Universal Robots PolyScope program: mouvements camera.urp

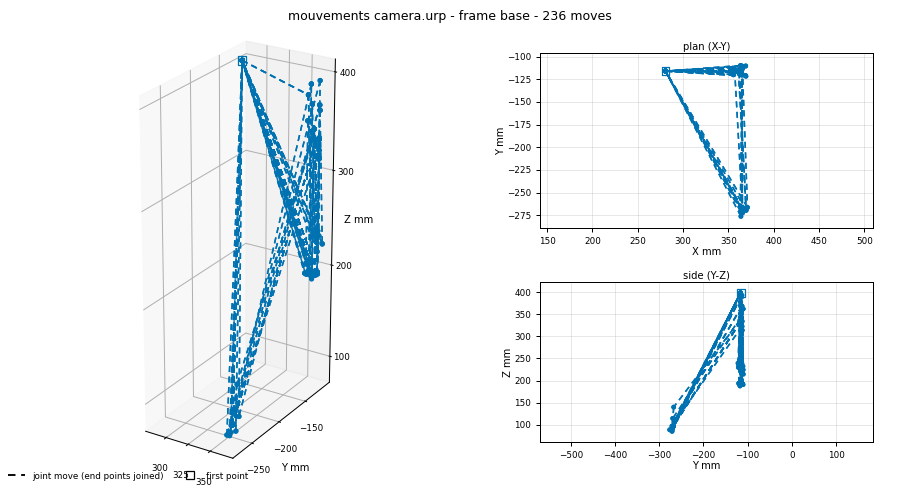
[picture p0: tool path of mouvements camera.urp in frame base, 236 of 236 moves have a stored position in this frame; points joined in program order, loops and branches not executed]
Program mouvements camera (installation=default directory=/programs/usbdisk_0 createdIn=5.21.2.0 lastSavedIn=5.12.2.1101534 robotSerialNumber=20185300595)
Calibrated DH parameters: a=[-0.000277, -0.17386, -0.213363, 0.000174, -0.000165, 0]; d=[0.151934, 52.001523, -51.96016, 0.089383, 0.08529, 0.092152]; alpha=[1.571075, 0.003287, -0.008212, 1.571169, -1.571801, 0]; deltaTheta=[0, 0.776939, 5.504669, 0.001575, 0, 0]
InitVariablesNode
Robot Program (runOnlyOnce=true)
  Folder Mouvements L'
    MoveJ speed 60 deg/s, acceleration 80 deg/s^2 (useActiveTCP=true) feature=Base
      Waypoint Waypoint_2: motionParameters(jointSpeed=1.047198 jointAcceleration=1.396263 cartesianSpeed=0.25 cartesianAcceleration=1.2); TCP in base x=280.608 y=-116.08 z=398.046 mm, rx=-2.2371 ry=2.1464 rz=-0.0359 rad; joints [2.971, -88.172, -66.4, 247.256, 90.066, 0.681] deg
      MoveJ speed 60 deg/s, acceleration 80 deg/s^2 (useActiveTCP=true) feature=Base
        Waypoint Waypoint_64: TCP in base x=354.47 y=-115.864 z=377.183 mm, rx=-3.1272 ry=-0.0242 rz=-0.0175 rad; joints [2.354, -105.869, -51.286, 247.88, 90.252, -88.495] deg
        MoveJ speed 60 deg/s, acceleration 80 deg/s^2 (useActiveTCP=true) feature=Base
          Waypoint Waypoint_65: TCP in base x=360.926 y=-115.109 z=191.362 mm, rx=-3.1273 ry=-0.0242 rz=-0.0173 rad; joints [2.478, -109.435, -98.039, 298.19, 90.28, -88.777] deg
          URCap Gripper (Robotiq_Grippers, Robotiq Inc.) dataModel(position=100.0, force=0.0, speed=0.0, positionInDouble=100.0, forceInDouble=0.0, speedInDouble=0.0, slaveIds=[2], blocking=true)
          MoveJ speed 60 deg/s, acceleration 80 deg/s^2 (useActiveTCP=true) feature=Base
            Waypoint Waypoint_66: TCP in base x=360.933 y=-115.105 z=343.669 mm, rx=-3.1273 ry=-0.0242 rz=-0.0174 rad; joints [2.446, -104.701, -62.277, 257.7, 90.221, -88.479] deg
            MoveJ speed 60 deg/s, acceleration 80 deg/s^2 (useActiveTCP=true) feature=Base
              Waypoint Waypoint_67: TCP in base x=360.932 y=-115.1 z=343.683 mm, rx=0.037 ry=-3.1303 rz=0.0223 rad; joints [2.853, -105.13, -61.17, 255.696, 88.644, 91.476] deg
              MoveJ speed 60 deg/s, acceleration 80 deg/s^2 (useActiveTCP=true) feature=Base
                Waypoint Waypoint_68: TCP in base x=369.453 y=-269.495 z=114.41 mm, rx=0.0346 ry=-2.5587 rz=-1.7903 rad; joints [-29.022, -179.68, 16.641, 199.059, 143.672, 30.692] deg
                MoveJ speed 60 deg/s, acceleration 80 deg/s^2 (useActiveTCP=true) feature=Base
                  Waypoint Waypoint_79: TCP in base x=369.462 y=-269.49 z=91.378 mm, rx=0.0347 ry=-2.5588 rz=-1.7903 rad; joints [-29.026, -184.503, 20.753, 199.764, 143.68, 30.679] deg
                URCap Gripper (Robotiq_Grippers, Robotiq Inc.) dataModel(position=0.0, force=0.0, speed=0.0, positionInDouble=0.0, forceInDouble=0.0, speedInDouble=0.0, slaveIds=[2], blocking=true)
                MoveJ speed 60 deg/s, acceleration 80 deg/s^2 (useActiveTCP=true) feature=Base
                  Waypoint Waypoint_2: motionParameters(jointSpeed=1.047198 jointAcceleration=1.396263 cartesianSpeed=0.25 cartesianAcceleration=1.2); TCP in base x=280.608 y=-116.08 z=398.046 mm, rx=-2.2371 ry=2.1464 rz=-0.0359 rad; joints [2.971, -88.172, -66.4, 247.256, 90.066, 0.681] deg
                  MoveJ speed 60 deg/s, acceleration 80 deg/s^2 (useActiveTCP=true) feature=Base
                    MoveJ speed 60 deg/s, acceleration 80 deg/s^2 (useActiveTCP=true) feature=Base
                      MoveJ speed 60 deg/s, acceleration 80 deg/s^2 (useActiveTCP=true) feature=Base
                        MoveJ speed 60 deg/s, acceleration 80 deg/s^2 (useActiveTCP=true) feature=Base
                          MoveJ speed 60 deg/s, acceleration 80 deg/s^2 (useActiveTCP=true) feature=Base
                            MoveJ speed 60 deg/s, acceleration 80 deg/s^2 (useActiveTCP=true) feature=Base
                              Waypoint Waypoint_73: TCP in base x=355.313 y=-120.114 z=193.384 mm, rx=-2.2194 ry=2.165 rz=-0.0363 rad; joints [1.736, -108.041, -100.308, 301.021, 90.164, -0.064] deg
                              URCap Gripper (Robotiq_Grippers, Robotiq Inc.) dataModel(position=100.0, force=0.0, speed=0.0, positionInDouble=100.0, forceInDouble=0.0, speedInDouble=0.0, slaveIds=[2], blocking=true)
                              MoveJ speed 60 deg/s, acceleration 80 deg/s^2 (useActiveTCP=true) feature=Base
                                Waypoint Waypoint_77: TCP in base x=355.961 y=-120.112 z=194.005 mm, rx=-3.0953 ry=0.0462 rz=0.0063 rad; joints [1.212, -108.815, -97.781, 296.498, 92.122, -87.439] deg
                                URCap Gripper (Robotiq_Grippers, Robotiq Inc.) dataModel(position=0.0, force=0.0, speed=0.0, positionInDouble=0.0, forceInDouble=0.0, speedInDouble=0.0, slaveIds=[2], blocking=true)
                                MoveJ speed 60 deg/s, acceleration 80 deg/s^2 (useActiveTCP=true) feature=Base
                                  Waypoint Waypoint_2: motionParameters(jointSpeed=1.047198 jointAcceleration=1.396263 cartesianSpeed=0.25 cartesianAcceleration=1.2); TCP in base x=280.608 y=-116.08 z=398.046 mm, rx=-2.2371 ry=2.1464 rz=-0.0359 rad; joints [2.971, -88.172, -66.4, 247.256, 90.066, 0.681] deg
                                  MoveJ speed 60 deg/s, acceleration 80 deg/s^2 (useActiveTCP=true) feature=Base
                                    Waypoint Waypoint_64: TCP in base x=354.47 y=-115.864 z=377.183 mm, rx=-3.1272 ry=-0.0242 rz=-0.0175 rad; joints [2.354, -105.869, -51.286, 247.88, 90.252, -88.495] deg
                                    MoveJ speed 60 deg/s, acceleration 80 deg/s^2 (useActiveTCP=true) feature=Base
                                      Waypoint Waypoint_65: TCP in base x=360.926 y=-115.109 z=191.362 mm, rx=-3.1273 ry=-0.0242 rz=-0.0173 rad; joints [2.478, -109.435, -98.039, 298.19, 90.28, -88.777] deg
                                      URCap Gripper (Robotiq_Grippers, Robotiq Inc.) dataModel(position=100.0, force=0.0, speed=0.0, positionInDouble=100.0, forceInDouble=0.0, speedInDouble=0.0, slaveIds=[2], blocking=true)
                                      MoveJ speed 60 deg/s, acceleration 80 deg/s^2 (useActiveTCP=true) feature=Base
                                        Waypoint Waypoint_66: TCP in base x=360.933 y=-115.105 z=343.669 mm, rx=-3.1273 ry=-0.0242 rz=-0.0174 rad; joints [2.446, -104.701, -62.277, 257.7, 90.221, -88.479] deg
                                        MoveJ speed 60 deg/s, acceleration 80 deg/s^2 (useActiveTCP=true) feature=Base
                                          Waypoint Waypoint_67: TCP in base x=360.932 y=-115.1 z=343.683 mm, rx=0.037 ry=-3.1303 rz=0.0223 rad; joints [2.853, -105.13, -61.17, 255.696, 88.644, 91.476] deg
                                          MoveJ speed 60 deg/s, acceleration 80 deg/s^2 (useActiveTCP=true) feature=Base
                                            Waypoint Waypoint_70: TCP in base x=369.313 y=-121.75 z=239.195 mm, rx=0.037 ry=-3.1302 rz=0.0223 rad; joints [1.772, -107.864, -85.879, 283.154, 88.636, 90.168] deg
                                            URCap Gripper (Robotiq_Grippers, Robotiq Inc.) dataModel(position=0.0, force=0.0, speed=0.0, positionInDouble=0.0, forceInDouble=0.0, speedInDouble=0.0, slaveIds=[2], blocking=true)
                                            MoveJ speed 60 deg/s, acceleration 80 deg/s^2 (useActiveTCP=true) feature=Base
                                              Waypoint Waypoint_2: motionParameters(jointSpeed=1.047198 jointAcceleration=1.396263 cartesianSpeed=0.25 cartesianAcceleration=1.2); TCP in base x=280.608 y=-116.08 z=398.046 mm, rx=-2.2371 ry=2.1464 rz=-0.0359 rad; joints [2.971, -88.172, -66.4, 247.256, 90.066, 0.681] deg
                                              MoveJ speed 60 deg/s, acceleration 80 deg/s^2 (useActiveTCP=true) feature=Base
                                                Waypoint Waypoint_71: TCP in base x=355.772 y=-117.714 z=191.403 mm, rx=-2.2393 ry=2.1483 rz=-0.0407 rad; joints [2.184, -108.169, -100.734, 301.575, 89.944, -0.582] deg
                                                URCap Gripper (Robotiq_Grippers, Robotiq Inc.) dataModel(position=100.0, force=0.0, speed=0.0, positionInDouble=100.0, forceInDouble=0.0, speedInDouble=0.0, slaveIds=[2], blocking=true)
                                                URCap Gripper (Robotiq_Grippers, Robotiq Inc.) dataModel(position=0.0, force=0.0, speed=0.0, positionInDouble=0.0, forceInDouble=0.0, speedInDouble=0.0, slaveIds=[2], blocking=true)
                                                MoveJ speed 60 deg/s, acceleration 80 deg/s^2 (useActiveTCP=true) feature=Base
                                                  Waypoint Waypoint_72: TCP in base x=361.681 y=-117.4 z=187.816 mm, rx=-3.1346 ry=0.019 rz=0.0078 rad; joints [2.202, -110.258, -97.51, 297.556, 89.9, -87.472] deg
                                                  URCap Gripper (Robotiq_Grippers, Robotiq Inc.) dataModel(position=100.0, force=0.0, speed=0.0, positionInDouble=100.0, forceInDouble=0.0, speedInDouble=0.0, slaveIds=[2], blocking=true)
                                                  MoveJ speed 60 deg/s, acceleration 80 deg/s^2 (useActiveTCP=true) feature=Base
                                                    Waypoint Waypoint_75: TCP in base x=361.669 y=-117.405 z=336.568 mm, rx=-3.1346 ry=0.0189 rz=0.0078 rad; joints [2.169, -105.101, -63.323, 258.214, 89.842, -87.187] deg
                                                    MoveJ speed 60 deg/s, acceleration 80 deg/s^2 (useActiveTCP=true) feature=Base
                                                      Waypoint Waypoint_76: TCP in base x=369.461 y=-267.242 z=139.99 mm, rx=-1.9057 ry=0.0195 rz=0.0548 rad; joints [-28.823, -170.798, 4.334, 201.346, 144.189, -147.418] deg
                                                      MoveJ speed 60 deg/s, acceleration 80 deg/s^2 (useActiveTCP=true) feature=Base
                                                        Waypoint Waypoint_78: TCP in base x=363.434 y=-271.007 z=85.521 mm, rx=-1.8332 ry=0.0118 rz=0.0275 rad; joints [-29.831, -179.351, 7.546, 200.182, 146.023, -154.193] deg
                                                        Waypoint Waypoint_78: TCP in base x=363.434 y=-271.007 z=85.521 mm, rx=-1.8332 ry=0.0118 rz=0.0275 rad; joints [-29.831, -179.351, 7.546, 200.182, 146.023, -154.193] deg
                                                      URCap Gripper (Robotiq_Grippers, Robotiq Inc.) dataModel(position=0.0, force=0.0, speed=0.0, positionInDouble=0.0, forceInDouble=0.0, speedInDouble=0.0, slaveIds=[2], blocking=true)
                                                      MoveJ speed 60 deg/s, acceleration 80 deg/s^2 (useActiveTCP=true) feature=Base
                                                        Waypoint Waypoint_2: motionParameters(jointSpeed=1.047198 jointAcceleration=1.396263 cartesianSpeed=0.25 cartesianAcceleration=1.2); TCP in base x=280.608 y=-116.08 z=398.046 mm, rx=-2.2371 ry=2.1464 rz=-0.0359 rad; joints [2.971, -88.172, -66.4, 247.256, 90.066, 0.681] deg
  Folder Mouvements L
    MoveJ speed 60 deg/s, acceleration 80 deg/s^2 (useActiveTCP=true) feature=Base
      Waypoint Waypoint_2: motionParameters(jointSpeed=1.047198 jointAcceleration=1.396263 cartesianSpeed=0.25 cartesianAcceleration=1.2); TCP in base x=280.608 y=-116.08 z=398.046 mm, rx=-2.2371 ry=2.1464 rz=-0.0359 rad; joints [2.971, -88.172, -66.4, 247.256, 90.066, 0.681] deg
      MoveJ speed 60 deg/s, acceleration 80 deg/s^2 (useActiveTCP=true) feature=Base
        Waypoint Waypoint_64: TCP in base x=354.47 y=-115.864 z=377.183 mm, rx=-3.1272 ry=-0.0242 rz=-0.0175 rad; joints [2.354, -105.869, -51.286, 247.88, 90.252, -88.495] deg
        MoveJ speed 60 deg/s, acceleration 80 deg/s^2 (useActiveTCP=true) feature=Base
          Waypoint Waypoint_65: TCP in base x=360.926 y=-115.109 z=191.362 mm, rx=-3.1273 ry=-0.0242 rz=-0.0173 rad; joints [2.478, -109.435, -98.039, 298.19, 90.28, -88.777] deg
          URCap Gripper (Robotiq_Grippers, Robotiq Inc.) dataModel(position=100.0, force=0.0, speed=0.0, positionInDouble=100.0, forceInDouble=0.0, speedInDouble=0.0, slaveIds=[2], blocking=true)
          MoveJ speed 60 deg/s, acceleration 80 deg/s^2 (useActiveTCP=true) feature=Base
            Waypoint Waypoint_66: TCP in base x=360.933 y=-115.105 z=343.669 mm, rx=-3.1273 ry=-0.0242 rz=-0.0174 rad; joints [2.446, -104.701, -62.277, 257.7, 90.221, -88.479] deg
            MoveJ speed 60 deg/s, acceleration 80 deg/s^2 (useActiveTCP=true) feature=Base
              Waypoint Waypoint_67: TCP in base x=360.932 y=-115.1 z=343.683 mm, rx=0.037 ry=-3.1303 rz=0.0223 rad; joints [2.853, -105.13, -61.17, 255.696, 88.644, 91.476] deg
              MoveJ speed 60 deg/s, acceleration 80 deg/s^2 (useActiveTCP=true) feature=Base
                Waypoint Waypoint_68: TCP in base x=369.453 y=-269.495 z=114.41 mm, rx=0.0346 ry=-2.5587 rz=-1.7903 rad; joints [-29.022, -179.68, 16.641, 199.059, 143.672, 30.692] deg
                MoveJ speed 60 deg/s, acceleration 80 deg/s^2 (useActiveTCP=true) feature=Base
                  Waypoint Waypoint_79: TCP in base x=369.462 y=-269.49 z=91.378 mm, rx=0.0347 ry=-2.5588 rz=-1.7903 rad; joints [-29.026, -184.503, 20.753, 199.764, 143.68, 30.679] deg
                URCap Gripper (Robotiq_Grippers, Robotiq Inc.) dataModel(position=0.0, force=0.0, speed=0.0, positionInDouble=0.0, forceInDouble=0.0, speedInDouble=0.0, slaveIds=[2], blocking=true)
                MoveJ speed 60 deg/s, acceleration 80 deg/s^2 (useActiveTCP=true) feature=Base
                  Waypoint Waypoint_2: motionParameters(jointSpeed=1.047198 jointAcceleration=1.396263 cartesianSpeed=0.25 cartesianAcceleration=1.2); TCP in base x=280.608 y=-116.08 z=398.046 mm, rx=-2.2371 ry=2.1464 rz=-0.0359 rad; joints [2.971, -88.172, -66.4, 247.256, 90.066, 0.681] deg
                  MoveJ speed 60 deg/s, acceleration 80 deg/s^2 (useActiveTCP=true) feature=Base
                    MoveJ speed 60 deg/s, acceleration 80 deg/s^2 (useActiveTCP=true) feature=Base
                      MoveJ speed 60 deg/s, acceleration 80 deg/s^2 (useActiveTCP=true) feature=Base
                        MoveJ speed 60 deg/s, acceleration 80 deg/s^2 (useActiveTCP=true) feature=Base
                          MoveJ speed 60 deg/s, acceleration 80 deg/s^2 (useActiveTCP=true) feature=Base
                            Waypoint Waypoint_2: motionParameters(jointSpeed=1.047198 jointAcceleration=1.396263 cartesianSpeed=0.25 cartesianAcceleration=1.2); TCP in base x=280.608 y=-116.08 z=398.046 mm, rx=-2.2371 ry=2.1464 rz=-0.0359 rad; joints [2.971, -88.172, -66.4, 247.256, 90.066, 0.681] deg
                            MoveJ speed 60 deg/s, acceleration 80 deg/s^2 (useActiveTCP=true) feature=Base
                              Waypoint Waypoint_73: TCP in base x=355.313 y=-120.114 z=193.384 mm, rx=-2.2194 ry=2.165 rz=-0.0363 rad; joints [1.736, -108.041, -100.308, 301.021, 90.164, -0.064] deg
                              URCap Gripper (Robotiq_Grippers, Robotiq Inc.) dataModel(position=100.0, force=0.0, speed=0.0, positionInDouble=100.0, forceInDouble=0.0, speedInDouble=0.0, slaveIds=[2], blocking=true)
                              MoveJ speed 60 deg/s, acceleration 80 deg/s^2 (useActiveTCP=true) feature=Base
                                Waypoint Waypoint_74: TCP in base x=354.955 y=-112.49 z=193.442 mm, rx=-0.1703 ry=3.1218 rz=-0.0705 rad; joints [3.842, -107.298, -100.501, 298.663, 86.895, 87.201] deg
                                URCap Gripper (Robotiq_Grippers, Robotiq Inc.) dataModel(position=0.0, force=0.0, speed=0.0, positionInDouble=0.0, forceInDouble=0.0, speedInDouble=0.0, slaveIds=[2], blocking=true)
                                MoveJ speed 60 deg/s, acceleration 80 deg/s^2 (useActiveTCP=true) feature=Base
                                  Waypoint Waypoint_2: motionParameters(jointSpeed=1.047198 jointAcceleration=1.396263 cartesianSpeed=0.25 cartesianAcceleration=1.2); TCP in base x=280.608 y=-116.08 z=398.046 mm, rx=-2.2371 ry=2.1464 rz=-0.0359 rad; joints [2.971, -88.172, -66.4, 247.256, 90.066, 0.681] deg
                                  MoveJ speed 60 deg/s, acceleration 80 deg/s^2 (useActiveTCP=true) feature=Base
                                    Waypoint Waypoint_64: TCP in base x=354.47 y=-115.864 z=377.183 mm, rx=-3.1272 ry=-0.0242 rz=-0.0175 rad; joints [2.354, -105.869, -51.286, 247.88, 90.252, -88.495] deg
                                    MoveJ speed 60 deg/s, acceleration 80 deg/s^2 (useActiveTCP=true) feature=Base
                                      Waypoint Waypoint_65: TCP in base x=360.926 y=-115.109 z=191.362 mm, rx=-3.1273 ry=-0.0242 rz=-0.0173 rad; joints [2.478, -109.435, -98.039, 298.19, 90.28, -88.777] deg
                                      URCap Gripper (Robotiq_Grippers, Robotiq Inc.) dataModel(position=100.0, force=0.0, speed=0.0, positionInDouble=100.0, forceInDouble=0.0, speedInDouble=0.0, slaveIds=[2], blocking=true)
                                      MoveJ speed 60 deg/s, acceleration 80 deg/s^2 (useActiveTCP=true) feature=Base
                                        Waypoint Waypoint_66: TCP in base x=360.933 y=-115.105 z=343.669 mm, rx=-3.1273 ry=-0.0242 rz=-0.0174 rad; joints [2.446, -104.701, -62.277, 257.7, 90.221, -88.479] deg
                                        MoveJ speed 60 deg/s, acceleration 80 deg/s^2 (useActiveTCP=true) feature=Base
                                          Waypoint Waypoint_67: TCP in base x=360.932 y=-115.1 z=343.683 mm, rx=0.037 ry=-3.1303 rz=0.0223 rad; joints [2.853, -105.13, -61.17, 255.696, 88.644, 91.476] deg
                                          MoveJ speed 60 deg/s, acceleration 80 deg/s^2 (useActiveTCP=true) feature=Base
                                            Waypoint Waypoint_70: TCP in base x=369.313 y=-121.75 z=239.195 mm, rx=0.037 ry=-3.1302 rz=0.0223 rad; joints [1.772, -107.864, -85.879, 283.154, 88.636, 90.168] deg
                                            URCap Gripper (Robotiq_Grippers, Robotiq Inc.) dataModel(position=0.0, force=0.0, speed=0.0, positionInDouble=0.0, forceInDouble=0.0, speedInDouble=0.0, slaveIds=[2], blocking=true)
                                            MoveJ speed 60 deg/s, acceleration 80 deg/s^2 (useActiveTCP=true) feature=Base
                                              Waypoint Waypoint_2: motionParameters(jointSpeed=1.047198 jointAcceleration=1.396263 cartesianSpeed=0.25 cartesianAcceleration=1.2); TCP in base x=280.608 y=-116.08 z=398.046 mm, rx=-2.2371 ry=2.1464 rz=-0.0359 rad; joints [2.971, -88.172, -66.4, 247.256, 90.066, 0.681] deg
                                              MoveJ speed 60 deg/s, acceleration 80 deg/s^2 (useActiveTCP=true) feature=Base
                                                Waypoint Waypoint_71: TCP in base x=355.772 y=-117.714 z=191.403 mm, rx=-2.2393 ry=2.1483 rz=-0.0407 rad; joints [2.184, -108.169, -100.734, 301.575, 89.944, -0.582] deg
                                                URCap Gripper (Robotiq_Grippers, Robotiq Inc.) dataModel(position=100.0, force=0.0, speed=0.0, positionInDouble=100.0, forceInDouble=0.0, speedInDouble=0.0, slaveIds=[2], blocking=true)
                                                URCap Gripper (Robotiq_Grippers, Robotiq Inc.) dataModel(position=0.0, force=0.0, speed=0.0, positionInDouble=0.0, forceInDouble=0.0, speedInDouble=0.0, slaveIds=[2], blocking=true)
                                                MoveJ speed 60 deg/s, acceleration 80 deg/s^2 (useActiveTCP=true) feature=Base
                                                  Waypoint Waypoint_72: TCP in base x=361.681 y=-117.4 z=187.816 mm, rx=-3.1346 ry=0.019 rz=0.0078 rad; joints [2.202, -110.258, -97.51, 297.556, 89.9, -87.472] deg
                                                  URCap Gripper (Robotiq_Grippers, Robotiq Inc.) dataModel(position=100.0, force=0.0, speed=0.0, positionInDouble=100.0, forceInDouble=0.0, speedInDouble=0.0, slaveIds=[2], blocking=true)
                                                  MoveJ speed 60 deg/s, acceleration 80 deg/s^2 (useActiveTCP=true) feature=Base
                                                    Waypoint Waypoint_75: TCP in base x=361.669 y=-117.405 z=336.568 mm, rx=-3.1346 ry=0.0189 rz=0.0078 rad; joints [2.169, -105.101, -63.323, 258.214, 89.842, -87.187] deg
                                                    MoveJ speed 60 deg/s, acceleration 80 deg/s^2 (useActiveTCP=true) feature=Base
                                                      Waypoint Waypoint_76: TCP in base x=369.461 y=-267.242 z=139.99 mm, rx=-1.9057 ry=0.0195 rz=0.0548 rad; joints [-28.823, -170.798, 4.334, 201.346, 144.189, -147.418] deg
                                                      MoveJ speed 60 deg/s, acceleration 80 deg/s^2 (useActiveTCP=true) feature=Base
                                                        Waypoint Waypoint_78: TCP in base x=363.434 y=-271.007 z=85.521 mm, rx=-1.8332 ry=0.0118 rz=0.0275 rad; joints [-29.831, -179.351, 7.546, 200.182, 146.023, -154.193] deg
                                                      URCap Gripper (Robotiq_Grippers, Robotiq Inc.) dataModel(position=0.0, force=0.0, speed=0.0, positionInDouble=0.0, forceInDouble=0.0, speedInDouble=0.0, slaveIds=[2], blocking=true)
                                                      MoveJ speed 60 deg/s, acceleration 80 deg/s^2 (useActiveTCP=true) feature=Base
                                                        Waypoint Waypoint_2: motionParameters(jointSpeed=1.047198 jointAcceleration=1.396263 cartesianSpeed=0.25 cartesianAcceleration=1.2); TCP in base x=280.608 y=-116.08 z=398.046 mm, rx=-2.2371 ry=2.1464 rz=-0.0359 rad; joints [2.971, -88.172, -66.4, 247.256, 90.066, 0.681] deg
  Folder Mouvement U
    MoveJ speed 60 deg/s, acceleration 80 deg/s^2 (useActiveTCP=true) feature=Base
      Waypoint Waypoint_2: motionParameters(jointSpeed=1.047198 jointAcceleration=1.396263 cartesianSpeed=0.25 cartesianAcceleration=1.2); TCP in base x=280.608 y=-116.08 z=398.046 mm, rx=-2.2371 ry=2.1464 rz=-0.0359 rad; joints [2.971, -88.172, -66.4, 247.256, 90.066, 0.681] deg
      MoveJ speed 60 deg/s, acceleration 80 deg/s^2 (useActiveTCP=true) feature=Base
        Waypoint Waypoint_8: TCP in base x=360.359 y=-116.083 z=194.377 mm, rx=-2.248 ry=2.1578 rz=0.0022 rad; joints [2.251, -109.03, -97.858, 297.936, 90.564, -0.456] deg
        URCap Gripper (Robotiq_Grippers, Robotiq Inc.) dataModel(position=100.0, force=0.0, speed=0.0, positionInDouble=100.0, forceInDouble=0.0, speedInDouble=0.0, slaveIds=[2], blocking=true)
        MoveJ speed 60 deg/s, acceleration 80 deg/s^2 (useActiveTCP=true) feature=Base
          Waypoint Waypoint_11: TCP in base x=360.347 y=-116.075 z=194.373 mm, rx=-0.1344 ry=3.1191 rz=-0.0257 rad; joints [2.778, -108.754, -98.304, 298.232, 88.541, 87.461] deg
          URCap Gripper (Robotiq_Grippers, Robotiq Inc.) dataModel(position=0.0, force=0.0, speed=0.0, positionInDouble=0.0, forceInDouble=0.0, speedInDouble=0.0, slaveIds=[2], blocking=true)
          MoveJ speed 60 deg/s, acceleration 80 deg/s^2 (useActiveTCP=true) feature=Base
            Waypoint Waypoint_2: motionParameters(jointSpeed=1.047198 jointAcceleration=1.396263 cartesianSpeed=0.25 cartesianAcceleration=1.2); TCP in base x=280.608 y=-116.08 z=398.046 mm, rx=-2.2371 ry=2.1464 rz=-0.0359 rad; joints [2.971, -88.172, -66.4, 247.256, 90.066, 0.681] deg
          Folder Mouvement U'
            MoveJ speed 60 deg/s, acceleration 80 deg/s^2 (useActiveTCP=true) feature=Base
              Waypoint Waypoint_2: motionParameters(jointSpeed=1.047198 jointAcceleration=1.396263 cartesianSpeed=0.25 cartesianAcceleration=1.2); TCP in base x=280.608 y=-116.08 z=398.046 mm, rx=-2.2371 ry=2.1464 rz=-0.0359 rad; joints [2.971, -88.172, -66.4, 247.256, 90.066, 0.681] deg
              MoveJ speed 60 deg/s, acceleration 80 deg/s^2 (useActiveTCP=true) feature=Base
                Waypoint Waypoint_13: TCP in base x=360.129 y=-115.918 z=194.945 mm, rx=-2.246 ry=2.1551 rz=-0.0175 rad; joints [2.383, -108.75, -98.377, 298.822, 90.174, -0.353] deg
                URCap Gripper (Robotiq_Grippers, Robotiq Inc.) dataModel(position=100.0, force=0.0, speed=0.0, positionInDouble=100.0, forceInDouble=0.0, speedInDouble=0.0, slaveIds=[2], blocking=true)
                MoveJ speed 60 deg/s, acceleration 80 deg/s^2 (useActiveTCP=true) feature=Base
                  Waypoint Waypoint_12: TCP in base x=360.146 y=-115.908 z=194.96 mm, rx=-3.1124 ry=-0.0686 rz=0.0193 rad; joints [2.131, -109.287, -96.569, 295.219, 91.114, -90.75] deg
                  URCap Gripper (Robotiq_Grippers, Robotiq Inc.) dataModel(position=0.0, force=0.0, speed=0.0, positionInDouble=0.0, forceInDouble=0.0, speedInDouble=0.0, slaveIds=[2], blocking=true)
                  Folder Mouvement F
                    MoveJ speed 60 deg/s, acceleration 80 deg/s^2 (useActiveTCP=true) feature=Base
                      Waypoint Waypoint_2: motionParameters(jointSpeed=1.047198 jointAcceleration=1.396263 cartesianSpeed=0.25 cartesianAcceleration=1.2); TCP in base x=280.608 y=-116.08 z=398.046 mm, rx=-2.2371 ry=2.1464 rz=-0.0359 rad; joints [2.971, -88.172, -66.4, 247.256, 90.066, 0.681] deg
                      MoveJ speed 60 deg/s, acceleration 80 deg/s^2 (useActiveTCP=true) feature=Base
                        Waypoint Waypoint_14: TCP in base x=365.369 y=-113.056 z=194.065 mm, rx=-2.2548 ry=2.1638 rz=0.001 rad; joints [2.803, -109.941, -96.5, 297.16, 90.168, 0.082] deg
                        URCap Gripper (Robotiq_Grippers, Robotiq Inc.) dataModel(position=100.0, force=0.0, speed=0.0, positionInDouble=100.0, forceInDouble=0.0, speedInDouble=0.0, slaveIds=[2], blocking=true)
                        MoveJ speed 60 deg/s, acceleration 80 deg/s^2 (useActiveTCP=true) feature=Base
                          Waypoint Waypoint_15: TCP in base x=365.367 y=-113.056 z=313.339 mm, rx=-2.2546 ry=2.1637 rz=0.001 rad; joints [2.778, -104.495, -70.787, 266.006, 90.105, 0.314] deg
                          MoveJ speed 60 deg/s, acceleration 80 deg/s^2 (useActiveTCP=true) feature=Base
                            Waypoint Waypoint_23: TCP in base x=365.372 y=-113.061 z=392.746 mm, rx=-3.1299 ry=0.0024 rz=0.0189 rad; joints [2.738, -112.179, -37.095, 238.673, 90.207, -87.085] deg
                          MoveJ speed 60 deg/s, acceleration 80 deg/s^2 (useActiveTCP=true) feature=Base
                            Waypoint Waypoint_16: TCP in base x=363.126 y=-264.93 z=106.645 mm, rx=-1.9305 ry=-0.0066 rz=-0.0141 rad; joints [-29.004, -157.4, -33.157, 229.064, 144.815, -147.561] deg
                            URCap Gripper (Robotiq_Grippers, Robotiq Inc.) dataModel(position=0.0, force=0.0, speed=0.0, positionInDouble=0.0, forceInDouble=0.0, speedInDouble=0.0, slaveIds=[2], blocking=true)
                            MoveJ speed 60 deg/s, acceleration 80 deg/s^2 (useActiveTCP=true) feature=Base
                              Waypoint Waypoint_2: motionParameters(jointSpeed=1.047198 jointAcceleration=1.396263 cartesianSpeed=0.25 cartesianAcceleration=1.2); TCP in base x=280.608 y=-116.08 z=398.046 mm, rx=-2.2371 ry=2.1464 rz=-0.0359 rad; joints [2.971, -88.172, -66.4, 247.256, 90.066, 0.681] deg
                              MoveJ speed 60 deg/s, acceleration 80 deg/s^2 (useActiveTCP=true) feature=Base
                                Waypoint Waypoint_17: TCP in base x=359.006 y=-116.088 z=193.011 mm, rx=-2.2371 ry=2.1464 rz=-0.0359 rad; joints [2.365, -108.587, -99.655, 300.918, 90.181, -0.384] deg
                                URCap Gripper (Robotiq_Grippers, Robotiq Inc.) dataModel(position=100.0, force=0.0, speed=0.0, positionInDouble=100.0, forceInDouble=0.0, speedInDouble=0.0, slaveIds=[2], blocking=true)
                                MoveJ speed 60 deg/s, acceleration 80 deg/s^2 (useActiveTCP=true) feature=Base
                                  Waypoint Waypoint_18: TCP in base x=359.004 y=-116.091 z=368.94 mm, rx=-2.2371 ry=2.1464 rz=-0.0359 rad; joints [2.326, -105.125, -55.5, 253.299, 90.124, -0.043] deg
                                  MoveJ speed 60 deg/s, acceleration 80 deg/s^2 (useActiveTCP=true) feature=Base
                                    Waypoint Waypoint_19: TCP in base x=359.011 y=-116.091 z=368.946 mm, rx=-3.0949 ry=-0.0873 rz=0.0203 rad; joints [1.817, -107.4, -51.023, 247.739, 92.062, -91.397] deg
                                    MoveJ speed 60 deg/s, acceleration 80 deg/s^2 (useActiveTCP=true) feature=Base
                                      Waypoint Waypoint_20: TCP in base x=366.237 y=-120.423 z=235.896 mm, rx=-3.0949 ry=-0.0874 rz=0.0204 rad; joints [1.134, -107.736, -86.938, 283.944, 92.035, -92.376] deg
                                      URCap Gripper (Robotiq_Grippers, Robotiq Inc.) dataModel(position=0.0, force=0.0, speed=0.0, positionInDouble=0.0, forceInDouble=0.0, speedInDouble=0.0, slaveIds=[2], blocking=true)
                                      MoveJ speed 60 deg/s, acceleration 80 deg/s^2 (useActiveTCP=true) feature=Base
                                        Waypoint Waypoint_2: motionParameters(jointSpeed=1.047198 jointAcceleration=1.396263 cartesianSpeed=0.25 cartesianAcceleration=1.2); TCP in base x=280.608 y=-116.08 z=398.046 mm, rx=-2.2371 ry=2.1464 rz=-0.0359 rad; joints [2.971, -88.172, -66.4, 247.256, 90.066, 0.681] deg
                                        MoveJ speed 60 deg/s, acceleration 80 deg/s^2 (useActiveTCP=true) feature=Base
                                          Waypoint Waypoint_21: TCP in base x=364.127 y=-117.777 z=193.293 mm, rx=-2.2569 ry=2.1661 rz=0.0165 rad; joints [1.986, -110.209, -96.105, 296.494, 90.452, -0.727] deg
                                          URCap Gripper (Robotiq_Grippers, Robotiq Inc.) dataModel(position=100.0, force=0.0, speed=0.0, positionInDouble=100.0, forceInDouble=0.0, speedInDouble=0.0, slaveIds=[2], blocking=true)
                                          MoveJ speed 60 deg/s, acceleration 80 deg/s^2 (useActiveTCP=true) feature=Base
                                            Waypoint Waypoint_32: TCP in base x=364.117 y=-117.792 z=193.289 mm, rx=-0.0015 ry=3.1247 rz=-0.0036 rad; joints [2.276, -109.92, -96.897, 297.836, 89.322, 91.847] deg
                                          MoveJ speed 60 deg/s, acceleration 80 deg/s^2 (useActiveTCP=true) feature=Base
                                            MoveJ speed 60 deg/s, acceleration 80 deg/s^2 (useActiveTCP=true) feature=Base
                                              Waypoint Waypoint_2: motionParameters(jointSpeed=1.047198 jointAcceleration=1.396263 cartesianSpeed=0.25 cartesianAcceleration=1.2); TCP in base x=280.608 y=-116.08 z=398.046 mm, rx=-2.2371 ry=2.1464 rz=-0.0359 rad; joints [2.971, -88.172, -66.4, 247.256, 90.066, 0.681] deg
                                              MoveJ speed 60 deg/s, acceleration 80 deg/s^2 (useActiveTCP=true) feature=Base
                                                Waypoint Waypoint_24: TCP in base x=356.858 y=-114.748 z=193.459 mm, rx=-2.237 ry=2.1464 rz=-0.0359 rad; joints [2.599, -107.985, -100.366, 301.027, 90.17, -0.146] deg
                                                URCap Gripper (Robotiq_Grippers, Robotiq Inc.) dataModel(position=100.0, force=0.0, speed=0.0, positionInDouble=100.0, forceInDouble=0.0, speedInDouble=0.0, slaveIds=[2], blocking=true)
                                                MoveJ speed 60 deg/s, acceleration 80 deg/s^2 (useActiveTCP=true) feature=Base
                                                  Waypoint Waypoint_25: TCP in base x=356.855 y=-114.738 z=388.235 mm, rx=-2.2372 ry=2.1464 rz=-0.0359 rad; joints [2.556, -106.57, -47.975, 247.22, 90.134, 0.231] deg
                                                  MoveJ speed 60 deg/s, acceleration 80 deg/s^2 (useActiveTCP=true) feature=Base
                                                    Waypoint Waypoint_27: TCP in base x=356.863 y=-114.749 z=388.208 mm, rx=-3.1012 ry=-0.0612 rz=0.0211 rad; joints [2.118, -109.149, -42.896, 241.364, 91.775, -90.078] deg
                                                  MoveJ speed 60 deg/s, acceleration 80 deg/s^2 (useActiveTCP=true) feature=Base
                                                    Waypoint Waypoint_26: TCP in base x=365.655 y=-272.422 z=90.213 mm, rx=-1.8494 ry=-0.0463 rz=-0.0141 rad; joints [-29.785, -175.347, 0.325, 204.9, 145.531, -156.47] deg
                                                    URCap Gripper (Robotiq_Grippers, Robotiq Inc.) dataModel(position=0.0, force=0.0, speed=0.0, positionInDouble=0.0, forceInDouble=0.0, speedInDouble=0.0, slaveIds=[2], blocking=true)
                                                    MoveJ speed 60 deg/s, acceleration 80 deg/s^2 (useActiveTCP=true) feature=Base
                                                      Waypoint Waypoint_2: motionParameters(jointSpeed=1.047198 jointAcceleration=1.396263 cartesianSpeed=0.25 cartesianAcceleration=1.2); TCP in base x=280.608 y=-116.08 z=398.046 mm, rx=-2.2371 ry=2.1464 rz=-0.0359 rad; joints [2.971, -88.172, -66.4, 247.256, 90.066, 0.681] deg
                                                      MoveJ speed 60 deg/s, acceleration 80 deg/s^2 (useActiveTCP=true) feature=Base
                                                        Waypoint Waypoint_28: TCP in base x=354.352 y=-116.082 z=201.505 mm, rx=-2.237 ry=2.1464 rz=-0.0359 rad; joints [2.395, -106.647, -99.774, 299.096, 90.165, -0.336] deg
                                                        URCap Gripper (Robotiq_Grippers, Robotiq Inc.) dataModel(position=100.0, force=0.0, speed=0.0, positionInDouble=100.0, forceInDouble=0.0, speedInDouble=0.0, slaveIds=[2], blocking=true)
                                                        MoveJ speed 60 deg/s, acceleration 80 deg/s^2 (useActiveTCP=true) feature=Base
                                                          Waypoint Waypoint_29: TCP in base x=354.342 y=-116.082 z=351.047 mm, rx=-2.2371 ry=2.1464 rz=-0.0359 rad; joints [2.364, -102.529, -63.836, 259.041, 90.104, -0.046] deg
                                                          MoveJ speed 60 deg/s, acceleration 80 deg/s^2 (useActiveTCP=true) feature=Base
                                                            Waypoint Waypoint_30: TCP in base x=354.353 y=-116.08 z=351.019 mm, rx=-3.0948 ry=-0.093 rz=0.0205 rad; joints [1.85, -104.53, -59.905, 253.739, 92.034, -91.617] deg
                                                            MoveJ speed 60 deg/s, acceleration 80 deg/s^2 (useActiveTCP=true) feature=Base
                                                              Waypoint Waypoint_31: TCP in base x=368.984 y=-120.916 z=229.682 mm, rx=-3.0957 ry=0.0142 rz=0.018 rad; joints [1.041, -108.753, -87.348, 285.539, 92.083, -88.72] deg
                                                              URCap Gripper (Robotiq_Grippers, Robotiq Inc.) dataModel(position=0.0, force=0.0, speed=0.0, positionInDouble=0.0, forceInDouble=0.0, speedInDouble=0.0, slaveIds=[2], blocking=true)
                                                              MoveJ speed 60 deg/s, acceleration 80 deg/s^2 (useActiveTCP=true) feature=Base
                                                                Waypoint Waypoint_2: motionParameters(jointSpeed=1.047198 jointAcceleration=1.396263 cartesianSpeed=0.25 cartesianAcceleration=1.2); TCP in base x=280.608 y=-116.08 z=398.046 mm, rx=-2.2371 ry=2.1464 rz=-0.0359 rad; joints [2.971, -88.172, -66.4, 247.256, 90.066, 0.681] deg
                  Folder Mouvement F'
                    MoveJ speed 60 deg/s, acceleration 80 deg/s^2 (useActiveTCP=true) feature=Base
                      Waypoint Waypoint_2: motionParameters(jointSpeed=1.047198 jointAcceleration=1.396263 cartesianSpeed=0.25 cartesianAcceleration=1.2); TCP in base x=280.608 y=-116.08 z=398.046 mm, rx=-2.2371 ry=2.1464 rz=-0.0359 rad; joints [2.971, -88.172, -66.4, 247.256, 90.066, 0.681] deg
                      MoveJ speed 60 deg/s, acceleration 80 deg/s^2 (useActiveTCP=true) feature=Base
                        Waypoint Waypoint_14: TCP in base x=365.369 y=-113.056 z=194.065 mm, rx=-2.2548 ry=2.1638 rz=0.001 rad; joints [2.803, -109.941, -96.5, 297.16, 90.168, 0.082] deg
                        URCap Gripper (Robotiq_Grippers, Robotiq Inc.) dataModel(position=100.0, force=0.0, speed=0.0, positionInDouble=100.0, forceInDouble=0.0, speedInDouble=0.0, slaveIds=[2], blocking=true)
                        MoveJ speed 60 deg/s, acceleration 80 deg/s^2 (useActiveTCP=true) feature=Base
                          Waypoint Waypoint_15: TCP in base x=365.367 y=-113.056 z=313.339 mm, rx=-2.2546 ry=2.1637 rz=0.001 rad; joints [2.778, -104.495, -70.787, 266.006, 90.105, 0.314] deg
                          MoveJ speed 60 deg/s, acceleration 80 deg/s^2 (useActiveTCP=true) feature=Base
                            Waypoint Waypoint_23: TCP in base x=365.372 y=-113.061 z=392.746 mm, rx=-3.1299 ry=0.0024 rz=0.0189 rad; joints [2.738, -112.179, -37.095, 238.673, 90.207, -87.085] deg
                          MoveJ speed 60 deg/s, acceleration 80 deg/s^2 (useActiveTCP=true) feature=Base
                            Waypoint Waypoint_16: TCP in base x=363.126 y=-264.93 z=106.645 mm, rx=-1.9305 ry=-0.0066 rz=-0.0141 rad; joints [-29.004, -157.4, -33.157, 229.064, 144.815, -147.561] deg
                            URCap Gripper (Robotiq_Grippers, Robotiq Inc.) dataModel(position=0.0, force=0.0, speed=0.0, positionInDouble=0.0, forceInDouble=0.0, speedInDouble=0.0, slaveIds=[2], blocking=true)
                            MoveJ speed 60 deg/s, acceleration 80 deg/s^2 (useActiveTCP=true) feature=Base
                              Waypoint Waypoint_2: motionParameters(jointSpeed=1.047198 jointAcceleration=1.396263 cartesianSpeed=0.25 cartesianAcceleration=1.2); TCP in base x=280.608 y=-116.08 z=398.046 mm, rx=-2.2371 ry=2.1464 rz=-0.0359 rad; joints [2.971, -88.172, -66.4, 247.256, 90.066, 0.681] deg
                              MoveJ speed 60 deg/s, acceleration 80 deg/s^2 (useActiveTCP=true) feature=Base
                                Waypoint Waypoint_17: TCP in base x=359.006 y=-116.088 z=193.011 mm, rx=-2.2371 ry=2.1464 rz=-0.0359 rad; joints [2.365, -108.587, -99.655, 300.918, 90.181, -0.384] deg
                                URCap Gripper (Robotiq_Grippers, Robotiq Inc.) dataModel(position=100.0, force=0.0, speed=0.0, positionInDouble=100.0, forceInDouble=0.0, speedInDouble=0.0, slaveIds=[2], blocking=true)
                                MoveJ speed 60 deg/s, acceleration 80 deg/s^2 (useActiveTCP=true) feature=Base
                                  Waypoint Waypoint_18: TCP in base x=359.004 y=-116.091 z=368.94 mm, rx=-2.2371 ry=2.1464 rz=-0.0359 rad; joints [2.326, -105.125, -55.5, 253.299, 90.124, -0.043] deg
                                  MoveJ speed 60 deg/s, acceleration 80 deg/s^2 (useActiveTCP=true) feature=Base
                                    Waypoint Waypoint_19: TCP in base x=359.011 y=-116.091 z=368.946 mm, rx=-3.0949 ry=-0.0873 rz=0.0203 rad; joints [1.817, -107.4, -51.023, 247.739, 92.062, -91.397] deg
                                    MoveJ speed 60 deg/s, acceleration 80 deg/s^2 (useActiveTCP=true) feature=Base
                                      Waypoint Waypoint_20: TCP in base x=366.237 y=-120.423 z=235.896 mm, rx=-3.0949 ry=-0.0874 rz=0.0204 rad; joints [1.134, -107.736, -86.938, 283.944, 92.035, -92.376] deg
                                      URCap Gripper (Robotiq_Grippers, Robotiq Inc.) dataModel(position=0.0, force=0.0, speed=0.0, positionInDouble=0.0, forceInDouble=0.0, speedInDouble=0.0, slaveIds=[2], blocking=true)
                                      MoveJ speed 60 deg/s, acceleration 80 deg/s^2 (useActiveTCP=true) feature=Base
                                        Waypoint Waypoint_2: motionParameters(jointSpeed=1.047198 jointAcceleration=1.396263 cartesianSpeed=0.25 cartesianAcceleration=1.2); TCP in base x=280.608 y=-116.08 z=398.046 mm, rx=-2.2371 ry=2.1464 rz=-0.0359 rad; joints [2.971, -88.172, -66.4, 247.256, 90.066, 0.681] deg
                                        MoveJ speed 60 deg/s, acceleration 80 deg/s^2 (useActiveTCP=true) feature=Base
                                          Waypoint Waypoint_21: TCP in base x=364.127 y=-117.777 z=193.293 mm, rx=-2.2569 ry=2.1661 rz=0.0165 rad; joints [1.986, -110.209, -96.105, 296.494, 90.452, -0.727] deg
                                          URCap Gripper (Robotiq_Grippers, Robotiq Inc.) dataModel(position=100.0, force=0.0, speed=0.0, positionInDouble=100.0, forceInDouble=0.0, speedInDouble=0.0, slaveIds=[2], blocking=true)
                                          MoveJ speed 60 deg/s, acceleration 80 deg/s^2 (useActiveTCP=true) feature=Base
                                            Waypoint Waypoint_22: TCP in base x=364.117 y=-117.783 z=193.288 mm, rx=-3.1392 ry=-0.0124 rz=0.0265 rad; joints [2.189, -110.312, -95.473, 294.88, 89.639, -88.615] deg
                                            URCap Gripper (Robotiq_Grippers, Robotiq Inc.) dataModel(position=0.0, force=0.0, speed=0.0, positionInDouble=0.0, forceInDouble=0.0, speedInDouble=0.0, slaveIds=[2], blocking=true)
                                          MoveJ speed 60 deg/s, acceleration 80 deg/s^2 (useActiveTCP=true) feature=Base
                                            MoveJ speed 60 deg/s, acceleration 80 deg/s^2 (useActiveTCP=true) feature=Base
                                              Waypoint Waypoint_2: motionParameters(jointSpeed=1.047198 jointAcceleration=1.396263 cartesianSpeed=0.25 cartesianAcceleration=1.2); TCP in base x=280.608 y=-116.08 z=398.046 mm, rx=-2.2371 ry=2.1464 rz=-0.0359 rad; joints [2.971, -88.172, -66.4, 247.256, 90.066, 0.681] deg
                                              MoveJ speed 60 deg/s, acceleration 80 deg/s^2 (useActiveTCP=true) feature=Base
                                                Waypoint Waypoint_24: TCP in base x=356.858 y=-114.748 z=193.459 mm, rx=-2.237 ry=2.1464 rz=-0.0359 rad; joints [2.599, -107.985, -100.366, 301.027, 90.17, -0.146] deg
                                                URCap Gripper (Robotiq_Grippers, Robotiq Inc.) dataModel(position=100.0, force=0.0, speed=0.0, positionInDouble=100.0, forceInDouble=0.0, speedInDouble=0.0, slaveIds=[2], blocking=true)
                                                MoveJ speed 60 deg/s, acceleration 80 deg/s^2 (useActiveTCP=true) feature=Base
                                                  Waypoint Waypoint_25: TCP in base x=356.855 y=-114.738 z=388.235 mm, rx=-2.2372 ry=2.1464 rz=-0.0359 rad; joints [2.556, -106.57, -47.975, 247.22, 90.134, 0.231] deg
                                                  MoveJ speed 60 deg/s, acceleration 80 deg/s^2 (useActiveTCP=true) feature=Base
                                                    Waypoint Waypoint_27: TCP in base x=356.863 y=-114.749 z=388.208 mm, rx=-3.1012 ry=-0.0612 rz=0.0211 rad; joints [2.118, -109.149, -42.896, 241.364, 91.775, -90.078] deg
                                                  MoveJ speed 60 deg/s, acceleration 80 deg/s^2 (useActiveTCP=true) feature=Base
                                                    Waypoint Waypoint_26: TCP in base x=365.655 y=-272.422 z=90.213 mm, rx=-1.8494 ry=-0.0463 rz=-0.0141 rad; joints [-29.785, -175.347, 0.325, 204.9, 145.531, -156.47] deg
                                                    URCap Gripper (Robotiq_Grippers, Robotiq Inc.) dataModel(position=0.0, force=0.0, speed=0.0, positionInDouble=0.0, forceInDouble=0.0, speedInDouble=0.0, slaveIds=[2], blocking=true)
                                                    MoveJ speed 60 deg/s, acceleration 80 deg/s^2 (useActiveTCP=true) feature=Base
                                                      Waypoint Waypoint_2: motionParameters(jointSpeed=1.047198 jointAcceleration=1.396263 cartesianSpeed=0.25 cartesianAcceleration=1.2); TCP in base x=280.608 y=-116.08 z=398.046 mm, rx=-2.2371 ry=2.1464 rz=-0.0359 rad; joints [2.971, -88.172, -66.4, 247.256, 90.066, 0.681] deg
                                                      MoveJ speed 60 deg/s, acceleration 80 deg/s^2 (useActiveTCP=true) feature=Base
                                                        Waypoint Waypoint_28: TCP in base x=354.352 y=-116.082 z=201.505 mm, rx=-2.237 ry=2.1464 rz=-0.0359 rad; joints [2.395, -106.647, -99.774, 299.096, 90.165, -0.336] deg
                                                        URCap Gripper (Robotiq_Grippers, Robotiq Inc.) dataModel(position=100.0, force=0.0, speed=0.0, positionInDouble=100.0, forceInDouble=0.0, speedInDouble=0.0, slaveIds=[2], blocking=true)
                                                        MoveJ speed 60 deg/s, acceleration 80 deg/s^2 (useActiveTCP=true) feature=Base
                                                          Waypoint Waypoint_29: TCP in base x=354.342 y=-116.082 z=351.047 mm, rx=-2.2371 ry=2.1464 rz=-0.0359 rad; joints [2.364, -102.529, -63.836, 259.041, 90.104, -0.046] deg
                                                          MoveJ speed 60 deg/s, acceleration 80 deg/s^2 (useActiveTCP=true) feature=Base
                                                            Waypoint Waypoint_30: TCP in base x=354.353 y=-116.08 z=351.019 mm, rx=-3.0948 ry=-0.093 rz=0.0205 rad; joints [1.85, -104.53, -59.905, 253.739, 92.034, -91.617] deg
                                                            MoveJ speed 60 deg/s, acceleration 80 deg/s^2 (useActiveTCP=true) feature=Base
                                                              Waypoint Waypoint_31: TCP in base x=368.984 y=-120.916 z=229.682 mm, rx=-3.0957 ry=0.0142 rz=0.018 rad; joints [1.041, -108.753, -87.348, 285.539, 92.083, -88.72] deg
                                                              URCap Gripper (Robotiq_Grippers, Robotiq Inc.) dataModel(position=0.0, force=0.0, speed=0.0, positionInDouble=0.0, forceInDouble=0.0, speedInDouble=0.0, slaveIds=[2], blocking=true)
                                                              MoveJ speed 60 deg/s, acceleration 80 deg/s^2 (useActiveTCP=true) feature=Base
                                                                Waypoint Waypoint_2: motionParameters(jointSpeed=1.047198 jointAcceleration=1.396263 cartesianSpeed=0.25 cartesianAcceleration=1.2); TCP in base x=280.608 y=-116.08 z=398.046 mm, rx=-2.2371 ry=2.1464 rz=-0.0359 rad; joints [2.971, -88.172, -66.4, 247.256, 90.066, 0.681] deg
                  Folder Mouvement B'
                    MoveJ speed 60 deg/s, acceleration 80 deg/s^2 (useActiveTCP=true) feature=Base
                      Waypoint Waypoint_2: motionParameters(jointSpeed=1.047198 jointAcceleration=1.396263 cartesianSpeed=0.25 cartesianAcceleration=1.2); TCP in base x=280.608 y=-116.08 z=398.046 mm, rx=-2.2371 ry=2.1464 rz=-0.0359 rad; joints [2.971, -88.172, -66.4, 247.256, 90.066, 0.681] deg
                      MoveJ speed 60 deg/s, acceleration 80 deg/s^2 (useActiveTCP=true) feature=Base
                        Waypoint Waypoint_14: TCP in base x=365.369 y=-113.056 z=194.065 mm, rx=-2.2548 ry=2.1638 rz=0.001 rad; joints [2.803, -109.941, -96.5, 297.16, 90.168, 0.082] deg
                        URCap Gripper (Robotiq_Grippers, Robotiq Inc.) dataModel(position=100.0, force=0.0, speed=0.0, positionInDouble=100.0, forceInDouble=0.0, speedInDouble=0.0, slaveIds=[2], blocking=true)
                      MoveJ speed 60 deg/s, acceleration 80 deg/s^2 (useActiveTCP=true) feature=Base
                        Waypoint Waypoint_15: TCP in base x=365.367 y=-113.056 z=313.339 mm, rx=-2.2546 ry=2.1637 rz=0.001 rad; joints [2.778, -104.495, -70.787, 266.006, 90.105, 0.314] deg
                        MoveJ speed 60 deg/s, acceleration 80 deg/s^2 (useActiveTCP=true) feature=Base
                          Waypoint Waypoint_33: TCP in base x=365.385 y=-113.047 z=368.046 mm, rx=-0.0821 ry=3.128 rz=-0.0172 rad; joints [3.104, -107.441, -51.812, 250.007, 88.808, 90.107] deg
                          MoveJ speed 60 deg/s, acceleration 80 deg/s^2 (useActiveTCP=true) feature=Base
                            Waypoint Waypoint_34: TCP in base x=363.742 y=-276.25 z=88.704 mm, rx=-0.0178 ry=2.5077 rz=1.8787 rad; joints [-30.329, -172.528, -6.113, 209.236, 145.611, 25.412] deg
                            URCap Gripper (Robotiq_Grippers, Robotiq Inc.) dataModel(position=0.0, force=0.0, speed=0.0, positionInDouble=0.0, forceInDouble=0.0, speedInDouble=0.0, slaveIds=[2], blocking=true)
                            MoveJ speed 60 deg/s, acceleration 80 deg/s^2 (useActiveTCP=true) feature=Base
                              Waypoint Waypoint_2: motionParameters(jointSpeed=1.047198 jointAcceleration=1.396263 cartesianSpeed=0.25 cartesianAcceleration=1.2); TCP in base x=280.608 y=-116.08 z=398.046 mm, rx=-2.2371 ry=2.1464 rz=-0.0359 rad; joints [2.971, -88.172, -66.4, 247.256, 90.066, 0.681] deg
                              MoveJ speed 60 deg/s, acceleration 80 deg/s^2 (useActiveTCP=true) feature=Base
                                Waypoint Waypoint_14: TCP in base x=365.369 y=-113.056 z=194.065 mm, rx=-2.2548 ry=2.1638 rz=0.001 rad; joints [2.803, -109.941, -96.5, 297.16, 90.168, 0.082] deg
                                URCap Gripper (Robotiq_Grippers, Robotiq Inc.) dataModel(position=100.0, force=0.0, speed=0.0, positionInDouble=100.0, forceInDouble=0.0, speedInDouble=0.0, slaveIds=[2], blocking=true)
                                MoveJ speed 60 deg/s, acceleration 80 deg/s^2 (useActiveTCP=true) feature=Base
                                  Waypoint Waypoint_15: TCP in base x=365.367 y=-113.056 z=313.339 mm, rx=-2.2546 ry=2.1637 rz=0.001 rad; joints [2.778, -104.495, -70.787, 266.006, 90.105, 0.314] deg
                                  MoveJ speed 60 deg/s, acceleration 80 deg/s^2 (useActiveTCP=true) feature=Base
                                    Waypoint Waypoint_35: TCP in base x=365.354 y=-113.066 z=314.963 mm, rx=-3.13 ry=-0.0087 rz=0.019 rad; joints [2.771, -105.106, -69.026, 263.525, 90.113, -87.642] deg
                                    MoveJ speed 60 deg/s, acceleration 80 deg/s^2 (useActiveTCP=true) feature=Base
                                      Waypoint Waypoint_36: TCP in base x=365.363 y=-113.054 z=238.209 mm, rx=-3.13 ry=-0.0088 rz=0.0188 rad; joints [2.788, -106.568, -87.895, 283.861, 90.13, -87.795] deg
                                      URCap Gripper (Robotiq_Grippers, Robotiq Inc.) dataModel(position=0.0, force=0.0, speed=0.0, positionInDouble=0.0, forceInDouble=0.0, speedInDouble=0.0, slaveIds=[2], blocking=true)
                                      MoveJ speed 60 deg/s, acceleration 80 deg/s^2 (useActiveTCP=true) feature=Base
                                        Waypoint Waypoint_37: TCP in base x=365.36 y=-113.056 z=193.806 mm, rx=-3.13 ry=-0.0088 rz=0.0188 rad; joints [2.797, -110.212, -95.598, 295.206, 90.172, -87.877] deg
                                        URCap Gripper (Robotiq_Grippers, Robotiq Inc.) dataModel(position=100.0, force=0.0, speed=0.0, positionInDouble=100.0, forceInDouble=0.0, speedInDouble=0.0, slaveIds=[2], blocking=true)
                                        MoveJ speed 60 deg/s, acceleration 80 deg/s^2 (useActiveTCP=true) feature=Base
                                          Waypoint Waypoint_38: TCP in base x=364.25 y=-113.557 z=190.832 mm, rx=2.2043 ry=2.2243 rz=-0.0489 rad; joints [3.318, -110.092, -96.543, 295.744, 87.873, -177.541] deg
                                          URCap Gripper (Robotiq_Grippers, Robotiq Inc.) dataModel(position=0.0, force=0.0, speed=0.0, positionInDouble=0.0, forceInDouble=0.0, speedInDouble=0.0, slaveIds=[2], blocking=true)
                                          MoveJ speed 60 deg/s, acceleration 80 deg/s^2 (useActiveTCP=true) feature=Base
                                            Waypoint Waypoint_39: TCP in base x=364.267 y=-110.422 z=190.857 mm, rx=2.2094 ry=2.2296 rz=-0.0374 rad; joints [3.666, -109.952, -96.743, 295.833, 88.467, -177.201] deg
                                            URCap Gripper (Robotiq_Grippers, Robotiq Inc.) dataModel(position=100.0, force=0.0, speed=0.0, positionInDouble=100.0, forceInDouble=0.0, speedInDouble=0.0, slaveIds=[2], blocking=true)
                                            MoveJ speed 60 deg/s, acceleration 80 deg/s^2 (useActiveTCP=true) feature=Base
                                              Waypoint Waypoint_40: TCP in base x=364.269 y=-110.435 z=361.887 mm, rx=2.2094 ry=2.2296 rz=-0.0374 rad; joints [3.624, -107.188, -53.229, 249.545, 88.441, -176.871] deg
                                              MoveJ speed 60 deg/s, acceleration 80 deg/s^2 (useActiveTCP=true) feature=Base
                                                Waypoint Waypoint_41: TCP in base x=364.266 y=-110.427 z=361.87 mm, rx=-3.1251 ry=-0.1058 rz=0.0299 rad; joints [3.143, -107.582, -52.635, 249.195, 90.312, -90.72] deg
                                                MoveJ speed 60 deg/s, acceleration 80 deg/s^2 (useActiveTCP=true) feature=Base
                                                  Waypoint Waypoint_42: TCP in base x=369.043 y=-110.425 z=224.327 mm, rx=-3.1263 ry=-0.0056 rz=0.0292 rad; joints [3.12, -108.275, -89.319, 286.625, 90.37, -87.375] deg
                                                  URCap Gripper (Robotiq_Grippers, Robotiq Inc.) dataModel(position=0.0, force=0.0, speed=0.0, positionInDouble=0.0, forceInDouble=0.0, speedInDouble=0.0, slaveIds=[2], blocking=true)
                                                  MoveJ speed 60 deg/s, acceleration 80 deg/s^2 (useActiveTCP=true) feature=Base
                                                    Waypoint Waypoint_2: motionParameters(jointSpeed=1.047198 jointAcceleration=1.396263 cartesianSpeed=0.25 cartesianAcceleration=1.2); TCP in base x=280.608 y=-116.08 z=398.046 mm, rx=-2.2371 ry=2.1464 rz=-0.0359 rad; joints [2.971, -88.172, -66.4, 247.256, 90.066, 0.681] deg
                                                    MoveJ speed 60 deg/s, acceleration 80 deg/s^2 (useActiveTCP=true) feature=Base
                                                      Waypoint Waypoint_14: motionParameters(jointSpeed=1.047198 jointAcceleration=1.396263 cartesianSpeed=0.25 cartesianAcceleration=1.2); TCP in base x=365.369 y=-113.056 z=194.065 mm, rx=-2.2548 ry=2.1638 rz=0.001 rad; joints [2.803, -109.941, -96.5, 297.16, 90.168, 0.082] deg
                                                      URCap Gripper (Robotiq_Grippers, Robotiq Inc.) dataModel(position=100.0, force=0.0, speed=0.0, positionInDouble=100.0, forceInDouble=0.0, speedInDouble=0.0, slaveIds=[2], blocking=true)
                                                      MoveJ speed 60 deg/s, acceleration 80 deg/s^2 (useActiveTCP=true) feature=Base
                                                        Waypoint Waypoint_43: TCP in base x=365.354 y=-113.064 z=322.295 mm, rx=-2.2548 ry=2.1638 rz=0.0011 rad; joints [2.775, -104.719, -68.078, 263.512, 90.105, 0.329] deg
                                                        MoveJ speed 60 deg/s, acceleration 80 deg/s^2 (useActiveTCP=true) feature=Base
                                                          Waypoint Waypoint_44: TCP in base x=365.37 y=-113.043 z=322.293 mm, rx=-3.1292 ry=-0.0866 rz=0.0193 rad; joints [2.782, -105.33, -66.741, 261.436, 90.078, -90.465] deg
                                                          MoveJ speed 60 deg/s, acceleration 80 deg/s^2 (useActiveTCP=true) feature=Base
                                                            Waypoint Waypoint_45: TCP in base x=365.392 y=-271.166 z=97.081 mm, rx=-1.8545 ry=-0.06 rz=-0.0266 rad; joints [-29.659, -170.062, -9.102, 209.69, 145.545, -156.821] deg
                                                            URCap Gripper (Robotiq_Grippers, Robotiq Inc.) dataModel(position=0.0, force=0.0, speed=0.0, positionInDouble=0.0, forceInDouble=0.0, speedInDouble=0.0, slaveIds=[2], blocking=true)
                                                            MoveJ speed 60 deg/s, acceleration 80 deg/s^2 (useActiveTCP=true) feature=Base
                                                              Waypoint Waypoint_2: motionParameters(jointSpeed=1.047198 jointAcceleration=1.396263 cartesianSpeed=0.25 cartesianAcceleration=1.2); TCP in base x=280.608 y=-116.08 z=398.046 mm, rx=-2.2371 ry=2.1464 rz=-0.0359 rad; joints [2.971, -88.172, -66.4, 247.256, 90.066, 0.681] deg
                                                              MoveJ speed 60 deg/s, acceleration 80 deg/s^2 (useActiveTCP=true) feature=Base
                                                                Waypoint Waypoint_14: motionParameters(jointSpeed=1.047198 jointAcceleration=1.396263 cartesianSpeed=0.25 cartesianAcceleration=1.2); TCP in base x=365.369 y=-113.056 z=194.065 mm, rx=-2.2548 ry=2.1638 rz=0.001 rad; joints [2.803, -109.941, -96.5, 297.16, 90.168, 0.082] deg
                                                                URCap Gripper (Robotiq_Grippers, Robotiq Inc.) dataModel(position=100.0, force=0.0, speed=0.0, positionInDouble=100.0, forceInDouble=0.0, speedInDouble=0.0, slaveIds=[2], blocking=true)
                                                                MoveJ speed 60 deg/s, acceleration 80 deg/s^2 (useActiveTCP=true) feature=Base
                                                                  Waypoint Waypoint_46: TCP in base x=365.359 y=-113.063 z=333.428 mm, rx=-2.2547 ry=2.1637 rz=0.001 rad; joints [2.772, -105.139, -64.514, 260.377, 90.11, 0.352] deg
                                                                  MoveJ speed 60 deg/s, acceleration 80 deg/s^2 (useActiveTCP=true) feature=Base
                                                                    Waypoint Waypoint_47: TCP in base x=365.371 y=-113.055 z=333.395 mm, rx=-3.1301 ry=-0.066 rz=0.0199 rad; joints [2.782, -105.8, -63.098, 258.244, 90.064, -89.685] deg
                                                                    MoveJ speed 60 deg/s, acceleration 80 deg/s^2 (useActiveTCP=true) feature=Base
                                                                      Waypoint Waypoint_48: TCP in base x=365.368 y=-110.776 z=232.224 mm, rx=-3.1301 ry=-0.066 rz=0.0199 rad; joints [3.167, -106.791, -89.245, 285.385, 90.078, -89.523] deg
                                                                      URCap Gripper (Robotiq_Grippers, Robotiq Inc.) dataModel(position=0.0, force=0.0, speed=0.0, positionInDouble=0.0, forceInDouble=0.0, speedInDouble=0.0, slaveIds=[2], blocking=true)
                                                                      MoveJ speed 60 deg/s, acceleration 80 deg/s^2 (useActiveTCP=true) feature=Base
                                                                        Waypoint Waypoint_2: motionParameters(jointSpeed=1.047198 jointAcceleration=1.396263 cartesianSpeed=0.25 cartesianAcceleration=1.2); TCP in base x=280.608 y=-116.08 z=398.046 mm, rx=-2.2371 ry=2.1464 rz=-0.0359 rad; joints [2.971, -88.172, -66.4, 247.256, 90.066, 0.681] deg
                                                                        MoveJ speed 60 deg/s, acceleration 80 deg/s^2 (useActiveTCP=true) feature=Base
                                                                          Waypoint Waypoint_52: TCP in base x=365.36 y=-113.081 z=194.065 mm, rx=-3.1296 ry=-0.0643 rz=0.0191 rad; joints [2.801, -110.187, -95.547, 295.109, 90.142, -89.906] deg
                                                                          URCap Gripper (Robotiq_Grippers, Robotiq Inc.) dataModel(position=100.0, force=0.0, speed=0.0, positionInDouble=100.0, forceInDouble=0.0, speedInDouble=0.0, slaveIds=[2], blocking=true)
                                                                          MoveJ speed 60 deg/s, acceleration 80 deg/s^2 (useActiveTCP=true) feature=Base
                                                                            Waypoint Waypoint_49: TCP in base x=365.357 y=-113.073 z=368.519 mm, rx=-3.1297 ry=-0.0643 rz=0.019 rad; joints [2.76, -108.552, -49.559, 247.491, 90.126, -89.565] deg
                                                                            MoveJ speed 60 deg/s, acceleration 80 deg/s^2 (useActiveTCP=true) feature=Base
                                                                              Waypoint Waypoint_50: TCP in base x=371.009 y=-266.422 z=106.052 mm, rx=-1.905 ry=-0.0309 rz=0.0365 rad; joints [-28.566, -166.397, -14.117, 214.916, 143.684, -150.284] deg
                                                                              URCap Gripper (Robotiq_Grippers, Robotiq Inc.) dataModel(position=0.0, force=0.0, speed=0.0, positionInDouble=0.0, forceInDouble=0.0, speedInDouble=0.0, slaveIds=[2], blocking=true)
                                                                              MoveJ speed 60 deg/s, acceleration 80 deg/s^2 (useActiveTCP=true) feature=Base
                                                                                Waypoint Waypoint_2: motionParameters(jointSpeed=1.047198 jointAcceleration=1.396263 cartesianSpeed=0.25 cartesianAcceleration=1.2); TCP in base x=280.608 y=-116.08 z=398.046 mm, rx=-2.2371 ry=2.1464 rz=-0.0359 rad; joints [2.971, -88.172, -66.4, 247.256, 90.066, 0.681] deg
                                                                                MoveJ speed 60 deg/s, acceleration 80 deg/s^2 (useActiveTCP=true) feature=Base
                                                                                  Waypoint Waypoint_14: motionParameters(jointSpeed=1.047198 jointAcceleration=1.396263 cartesianSpeed=0.25 cartesianAcceleration=1.2); TCP in base x=365.369 y=-113.056 z=194.065 mm, rx=-2.2548 ry=2.1638 rz=0.001 rad; joints [2.803, -109.941, -96.5, 297.16, 90.168, 0.082] deg
                                                                                  URCap Gripper (Robotiq_Grippers, Robotiq Inc.) dataModel(position=100.0, force=0.0, speed=0.0, positionInDouble=100.0, forceInDouble=0.0, speedInDouble=0.0, slaveIds=[2], blocking=true)
                                                                                  MoveJ speed 60 deg/s, acceleration 80 deg/s^2 (useActiveTCP=true) feature=Base
                                                                                    Waypoint Waypoint_51: TCP in base x=365.366 y=-113.068 z=335.109 mm, rx=-2.2547 ry=2.1638 rz=0.001 rad; joints [2.771, -105.221, -63.946, 259.888, 90.11, 0.356] deg
                                                                                    MoveJ speed 60 deg/s, acceleration 80 deg/s^2 (useActiveTCP=true) feature=Base
                                                                                      Waypoint Waypoint_53: TCP in base x=363.19 y=-109.909 z=214.454 mm, rx=2.2026 ry=2.2394 rz=-0.0262 rad; joints [3.662, -107.405, -93.459, 290.23, 88.801, -177.591] deg
                                                                                      URCap Gripper (Robotiq_Grippers, Robotiq Inc.) dataModel(position=0.0, force=0.0, speed=0.0, positionInDouble=0.0, forceInDouble=0.0, speedInDouble=0.0, slaveIds=[2], blocking=true)
                                                                                      MoveJ speed 60 deg/s, acceleration 80 deg/s^2 (useActiveTCP=true) feature=Base
                                                                                        Waypoint Waypoint_2: motionParameters(jointSpeed=1.047198 jointAcceleration=1.396263 cartesianSpeed=0.25 cartesianAcceleration=1.2); TCP in base x=280.608 y=-116.08 z=398.046 mm, rx=-2.2371 ry=2.1464 rz=-0.0359 rad; joints [2.971, -88.172, -66.4, 247.256, 90.066, 0.681] deg
                  Folder Mouvement B
                    MoveJ speed 60 deg/s, acceleration 80 deg/s^2 (useActiveTCP=true) feature=Base
                      Waypoint Waypoint_2: motionParameters(jointSpeed=1.047198 jointAcceleration=1.396263 cartesianSpeed=0.25 cartesianAcceleration=1.2); TCP in base x=280.608 y=-116.08 z=398.046 mm, rx=-2.2371 ry=2.1464 rz=-0.0359 rad; joints [2.971, -88.172, -66.4, 247.256, 90.066, 0.681] deg
                      MoveJ speed 60 deg/s, acceleration 80 deg/s^2 (useActiveTCP=true) feature=Base
                        Waypoint Waypoint_14: TCP in base x=365.369 y=-113.056 z=194.065 mm, rx=-2.2548 ry=2.1638 rz=0.001 rad; joints [2.803, -109.941, -96.5, 297.16, 90.168, 0.082] deg
                        URCap Gripper (Robotiq_Grippers, Robotiq Inc.) dataModel(position=100.0, force=0.0, speed=0.0, positionInDouble=100.0, forceInDouble=0.0, speedInDouble=0.0, slaveIds=[2], blocking=true)
                      MoveJ speed 60 deg/s, acceleration 80 deg/s^2 (useActiveTCP=true) feature=Base
                        Waypoint Waypoint_15: TCP in base x=365.367 y=-113.056 z=313.339 mm, rx=-2.2546 ry=2.1637 rz=0.001 rad; joints [2.778, -104.495, -70.787, 266.006, 90.105, 0.314] deg
                        MoveJ speed 60 deg/s, acceleration 80 deg/s^2 (useActiveTCP=true) feature=Base
                          Waypoint Waypoint_33: TCP in base x=365.385 y=-113.047 z=368.046 mm, rx=-0.0821 ry=3.128 rz=-0.0172 rad; joints [3.104, -107.441, -51.812, 250.007, 88.808, 90.107] deg
                          MoveJ speed 60 deg/s, acceleration 80 deg/s^2 (useActiveTCP=true) feature=Base
                            Waypoint Waypoint_34: TCP in base x=363.742 y=-276.25 z=88.704 mm, rx=-0.0178 ry=2.5077 rz=1.8787 rad; joints [-30.329, -172.528, -6.113, 209.236, 145.611, 25.412] deg
                            URCap Gripper (Robotiq_Grippers, Robotiq Inc.) dataModel(position=0.0, force=0.0, speed=0.0, positionInDouble=0.0, forceInDouble=0.0, speedInDouble=0.0, slaveIds=[2], blocking=true)
                            MoveJ speed 60 deg/s, acceleration 80 deg/s^2 (useActiveTCP=true) feature=Base
                              Waypoint Waypoint_2: motionParameters(jointSpeed=1.047198 jointAcceleration=1.396263 cartesianSpeed=0.25 cartesianAcceleration=1.2); TCP in base x=280.608 y=-116.08 z=398.046 mm, rx=-2.2371 ry=2.1464 rz=-0.0359 rad; joints [2.971, -88.172, -66.4, 247.256, 90.066, 0.681] deg
                              MoveJ speed 60 deg/s, acceleration 80 deg/s^2 (useActiveTCP=true) feature=Base
                                Waypoint Waypoint_14: TCP in base x=365.369 y=-113.056 z=194.065 mm, rx=-2.2548 ry=2.1638 rz=0.001 rad; joints [2.803, -109.941, -96.5, 297.16, 90.168, 0.082] deg
                                URCap Gripper (Robotiq_Grippers, Robotiq Inc.) dataModel(position=100.0, force=0.0, speed=0.0, positionInDouble=100.0, forceInDouble=0.0, speedInDouble=0.0, slaveIds=[2], blocking=true)
                                MoveJ speed 60 deg/s, acceleration 80 deg/s^2 (useActiveTCP=true) feature=Base
                                  Waypoint Waypoint_15: TCP in base x=365.367 y=-113.056 z=313.339 mm, rx=-2.2546 ry=2.1637 rz=0.001 rad; joints [2.778, -104.495, -70.787, 266.006, 90.105, 0.314] deg
                                  MoveJ speed 60 deg/s, acceleration 80 deg/s^2 (useActiveTCP=true) feature=Base
                                    Waypoint Waypoint_35: TCP in base x=365.354 y=-113.066 z=314.963 mm, rx=-3.13 ry=-0.0087 rz=0.019 rad; joints [2.771, -105.106, -69.026, 263.525, 90.113, -87.642] deg
                                    MoveJ speed 60 deg/s, acceleration 80 deg/s^2 (useActiveTCP=true) feature=Base
                                      Waypoint Waypoint_36: TCP in base x=365.363 y=-113.054 z=238.209 mm, rx=-3.13 ry=-0.0088 rz=0.0188 rad; joints [2.788, -106.568, -87.895, 283.861, 90.13, -87.795] deg
                                      URCap Gripper (Robotiq_Grippers, Robotiq Inc.) dataModel(position=0.0, force=0.0, speed=0.0, positionInDouble=0.0, forceInDouble=0.0, speedInDouble=0.0, slaveIds=[2], blocking=true)
                                      MoveJ speed 60 deg/s, acceleration 80 deg/s^2 (useActiveTCP=true) feature=Base
                                        Waypoint Waypoint_37: TCP in base x=365.36 y=-113.056 z=193.806 mm, rx=-3.13 ry=-0.0088 rz=0.0188 rad; joints [2.797, -110.212, -95.598, 295.206, 90.172, -87.877] deg
                                        URCap Gripper (Robotiq_Grippers, Robotiq Inc.) dataModel(position=100.0, force=0.0, speed=0.0, positionInDouble=100.0, forceInDouble=0.0, speedInDouble=0.0, slaveIds=[2], blocking=true)
                                        MoveJ speed 60 deg/s, acceleration 80 deg/s^2 (useActiveTCP=true) feature=Base
                                          Waypoint Waypoint_54: TCP in base x=365.365 y=-113.047 z=193.804 mm, rx=-2.1473 ry=2.2703 rz=-0.0003 rad; joints [2.822, -109.947, -96.599, 297.333, 90.104, 5.647] deg
                                          URCap Gripper (Robotiq_Grippers, Robotiq Inc.) dataModel(position=0.0, force=0.0, speed=0.0, positionInDouble=0.0, forceInDouble=0.0, speedInDouble=0.0, slaveIds=[2], blocking=true)
                                          MoveJ speed 60 deg/s, acceleration 80 deg/s^2 (useActiveTCP=true) feature=Base
                                            Waypoint Waypoint_39: TCP in base x=364.267 y=-110.422 z=190.857 mm, rx=2.2094 ry=2.2296 rz=-0.0374 rad; joints [3.666, -109.952, -96.743, 295.833, 88.467, -177.201] deg
                                            URCap Gripper (Robotiq_Grippers, Robotiq Inc.) dataModel(position=100.0, force=0.0, speed=0.0, positionInDouble=100.0, forceInDouble=0.0, speedInDouble=0.0, slaveIds=[2], blocking=true)
                                            MoveJ speed 60 deg/s, acceleration 80 deg/s^2 (useActiveTCP=true) feature=Base
                                              Waypoint Waypoint_40: TCP in base x=364.269 y=-110.435 z=361.887 mm, rx=2.2094 ry=2.2296 rz=-0.0374 rad; joints [3.624, -107.188, -53.229, 249.545, 88.441, -176.871] deg
                                              MoveJ speed 60 deg/s, acceleration 80 deg/s^2 (useActiveTCP=true) feature=Base
                                                Waypoint Waypoint_41: TCP in base x=364.266 y=-110.427 z=361.87 mm, rx=-3.1251 ry=-0.1058 rz=0.0299 rad; joints [3.143, -107.582, -52.635, 249.195, 90.312, -90.72] deg
                                                MoveJ speed 60 deg/s, acceleration 80 deg/s^2 (useActiveTCP=true) feature=Base
                                                  Waypoint Waypoint_42: TCP in base x=369.043 y=-110.425 z=224.327 mm, rx=-3.1263 ry=-0.0056 rz=0.0292 rad; joints [3.12, -108.275, -89.319, 286.625, 90.37, -87.375] deg
                                                  URCap Gripper (Robotiq_Grippers, Robotiq Inc.) dataModel(position=0.0, force=0.0, speed=0.0, positionInDouble=0.0, forceInDouble=0.0, speedInDouble=0.0, slaveIds=[2], blocking=true)
                                                  MoveJ speed 60 deg/s, acceleration 80 deg/s^2 (useActiveTCP=true) feature=Base
                                                    Waypoint Waypoint_55: TCP in base x=369.046 y=-110.42 z=224.328 mm, rx=-2.2576 ry=2.1504 rz=0.0056 rad; joints [3.083, -107.829, -90.718, 289.45, 90.541, 0] deg
                                                  MoveJ speed 60 deg/s, acceleration 80 deg/s^2 (useActiveTCP=true) feature=Base
                                                    Waypoint Waypoint_2: motionParameters(jointSpeed=1.047198 jointAcceleration=1.396263 cartesianSpeed=0.25 cartesianAcceleration=1.2); TCP in base x=280.608 y=-116.08 z=398.046 mm, rx=-2.2371 ry=2.1464 rz=-0.0359 rad; joints [2.971, -88.172, -66.4, 247.256, 90.066, 0.681] deg
                                                    MoveJ speed 60 deg/s, acceleration 80 deg/s^2 (useActiveTCP=true) feature=Base
                                                      Waypoint Waypoint_14: motionParameters(jointSpeed=1.047198 jointAcceleration=1.396263 cartesianSpeed=0.25 cartesianAcceleration=1.2); TCP in base x=365.369 y=-113.056 z=194.065 mm, rx=-2.2548 ry=2.1638 rz=0.001 rad; joints [2.803, -109.941, -96.5, 297.16, 90.168, 0.082] deg
                                                      URCap Gripper (Robotiq_Grippers, Robotiq Inc.) dataModel(position=100.0, force=0.0, speed=0.0, positionInDouble=100.0, forceInDouble=0.0, speedInDouble=0.0, slaveIds=[2], blocking=true)
                                                      MoveJ speed 60 deg/s, acceleration 80 deg/s^2 (useActiveTCP=true) feature=Base
                                                        Waypoint Waypoint_43: TCP in base x=365.354 y=-113.064 z=322.295 mm, rx=-2.2548 ry=2.1638 rz=0.0011 rad; joints [2.775, -104.719, -68.078, 263.512, 90.105, 0.329] deg
                                                        MoveJ speed 60 deg/s, acceleration 80 deg/s^2 (useActiveTCP=true) feature=Base
                                                          Waypoint Waypoint_44: TCP in base x=365.37 y=-113.043 z=322.293 mm, rx=-3.1292 ry=-0.0866 rz=0.0193 rad; joints [2.782, -105.33, -66.741, 261.436, 90.078, -90.465] deg
                                                          MoveJ speed 60 deg/s, acceleration 80 deg/s^2 (useActiveTCP=true) feature=Base
                                                            Waypoint Waypoint_45: TCP in base x=365.392 y=-271.166 z=97.081 mm, rx=-1.8545 ry=-0.06 rz=-0.0266 rad; joints [-29.659, -170.062, -9.102, 209.69, 145.545, -156.821] deg
                                                            URCap Gripper (Robotiq_Grippers, Robotiq Inc.) dataModel(position=0.0, force=0.0, speed=0.0, positionInDouble=0.0, forceInDouble=0.0, speedInDouble=0.0, slaveIds=[2], blocking=true)
                                                            MoveJ speed 60 deg/s, acceleration 80 deg/s^2 (useActiveTCP=true) feature=Base
                                                              Waypoint Waypoint_2: motionParameters(jointSpeed=1.047198 jointAcceleration=1.396263 cartesianSpeed=0.25 cartesianAcceleration=1.2); TCP in base x=280.608 y=-116.08 z=398.046 mm, rx=-2.2371 ry=2.1464 rz=-0.0359 rad; joints [2.971, -88.172, -66.4, 247.256, 90.066, 0.681] deg
                                                              MoveJ speed 60 deg/s, acceleration 80 deg/s^2 (useActiveTCP=true) feature=Base
                                                                Waypoint Waypoint_14: motionParameters(jointSpeed=1.047198 jointAcceleration=1.396263 cartesianSpeed=0.25 cartesianAcceleration=1.2); TCP in base x=365.369 y=-113.056 z=194.065 mm, rx=-2.2548 ry=2.1638 rz=0.001 rad; joints [2.803, -109.941, -96.5, 297.16, 90.168, 0.082] deg
                                                                URCap Gripper (Robotiq_Grippers, Robotiq Inc.) dataModel(position=100.0, force=0.0, speed=0.0, positionInDouble=100.0, forceInDouble=0.0, speedInDouble=0.0, slaveIds=[2], blocking=true)
                                                                MoveJ speed 60 deg/s, acceleration 80 deg/s^2 (useActiveTCP=true) feature=Base
                                                                  Waypoint Waypoint_46: TCP in base x=365.359 y=-113.063 z=333.428 mm, rx=-2.2547 ry=2.1637 rz=0.001 rad; joints [2.772, -105.139, -64.514, 260.377, 90.11, 0.352] deg
                                                                  MoveJ speed 60 deg/s, acceleration 80 deg/s^2 (useActiveTCP=true) feature=Base
                                                                    Waypoint Waypoint_47: TCP in base x=365.371 y=-113.055 z=333.395 mm, rx=-3.1301 ry=-0.066 rz=0.0199 rad; joints [2.782, -105.8, -63.098, 258.244, 90.064, -89.685] deg
                                                                    MoveJ speed 60 deg/s, acceleration 80 deg/s^2 (useActiveTCP=true) feature=Base
                                                                      Waypoint Waypoint_48: TCP in base x=365.368 y=-110.776 z=232.224 mm, rx=-3.1301 ry=-0.066 rz=0.0199 rad; joints [3.167, -106.791, -89.245, 285.385, 90.078, -89.523] deg
                                                                      URCap Gripper (Robotiq_Grippers, Robotiq Inc.) dataModel(position=0.0, force=0.0, speed=0.0, positionInDouble=0.0, forceInDouble=0.0, speedInDouble=0.0, slaveIds=[2], blocking=true)
                                                                      MoveJ speed 60 deg/s, acceleration 80 deg/s^2 (useActiveTCP=true) feature=Base
                                                                        Waypoint Waypoint_2: motionParameters(jointSpeed=1.047198 jointAcceleration=1.396263 cartesianSpeed=0.25 cartesianAcceleration=1.2); TCP in base x=280.608 y=-116.08 z=398.046 mm, rx=-2.2371 ry=2.1464 rz=-0.0359 rad; joints [2.971, -88.172, -66.4, 247.256, 90.066, 0.681] deg
                                                                        MoveJ speed 60 deg/s, acceleration 80 deg/s^2 (useActiveTCP=true) feature=Base
                                                                          Waypoint Waypoint_52: TCP in base x=365.36 y=-113.081 z=194.065 mm, rx=-3.1296 ry=-0.0643 rz=0.0191 rad; joints [2.801, -110.187, -95.547, 295.109, 90.142, -89.906] deg
                                                                          URCap Gripper (Robotiq_Grippers, Robotiq Inc.) dataModel(position=100.0, force=0.0, speed=0.0, positionInDouble=100.0, forceInDouble=0.0, speedInDouble=0.0, slaveIds=[2], blocking=true)
                                                                          MoveJ speed 60 deg/s, acceleration 80 deg/s^2 (useActiveTCP=true) feature=Base
                                                                            Waypoint Waypoint_49: TCP in base x=365.357 y=-113.073 z=368.519 mm, rx=-3.1297 ry=-0.0643 rz=0.019 rad; joints [2.76, -108.552, -49.559, 247.491, 90.126, -89.565] deg
                                                                            MoveJ speed 60 deg/s, acceleration 80 deg/s^2 (useActiveTCP=true) feature=Base
                                                                              Waypoint Waypoint_50: TCP in base x=371.009 y=-266.422 z=106.052 mm, rx=-1.905 ry=-0.0309 rz=0.0365 rad; joints [-28.566, -166.397, -14.117, 214.916, 143.684, -150.284] deg
                                                                              URCap Gripper (Robotiq_Grippers, Robotiq Inc.) dataModel(position=0.0, force=0.0, speed=0.0, positionInDouble=0.0, forceInDouble=0.0, speedInDouble=0.0, slaveIds=[2], blocking=true)
                                                                              MoveJ speed 60 deg/s, acceleration 80 deg/s^2 (useActiveTCP=true) feature=Base
                                                                                Waypoint Waypoint_2: motionParameters(jointSpeed=1.047198 jointAcceleration=1.396263 cartesianSpeed=0.25 cartesianAcceleration=1.2); TCP in base x=280.608 y=-116.08 z=398.046 mm, rx=-2.2371 ry=2.1464 rz=-0.0359 rad; joints [2.971, -88.172, -66.4, 247.256, 90.066, 0.681] deg
                                                                                MoveJ speed 60 deg/s, acceleration 80 deg/s^2 (useActiveTCP=true) feature=Base
                                                                                  Waypoint Waypoint_14: motionParameters(jointSpeed=1.047198 jointAcceleration=1.396263 cartesianSpeed=0.25 cartesianAcceleration=1.2); TCP in base x=365.369 y=-113.056 z=194.065 mm, rx=-2.2548 ry=2.1638 rz=0.001 rad; joints [2.803, -109.941, -96.5, 297.16, 90.168, 0.082] deg
                                                                                  URCap Gripper (Robotiq_Grippers, Robotiq Inc.) dataModel(position=100.0, force=0.0, speed=0.0, positionInDouble=100.0, forceInDouble=0.0, speedInDouble=0.0, slaveIds=[2], blocking=true)
                                                                                  MoveJ speed 60 deg/s, acceleration 80 deg/s^2 (useActiveTCP=true) feature=Base
                                                                                    Waypoint Waypoint_51: TCP in base x=365.366 y=-113.068 z=335.109 mm, rx=-2.2547 ry=2.1638 rz=0.001 rad; joints [2.771, -105.221, -63.946, 259.888, 90.11, 0.356] deg
                                                                                    MoveJ speed 60 deg/s, acceleration 80 deg/s^2 (useActiveTCP=true) feature=Base
                                                                                      Waypoint Waypoint_53: TCP in base x=363.19 y=-109.909 z=214.454 mm, rx=2.2026 ry=2.2394 rz=-0.0262 rad; joints [3.662, -107.405, -93.459, 290.23, 88.801, -177.591] deg
                                                                                      URCap Gripper (Robotiq_Grippers, Robotiq Inc.) dataModel(position=0.0, force=0.0, speed=0.0, positionInDouble=0.0, forceInDouble=0.0, speedInDouble=0.0, slaveIds=[2], blocking=true)
                                                                                      MoveJ speed 60 deg/s, acceleration 80 deg/s^2 (useActiveTCP=true) feature=Base
                                                                                        Waypoint Waypoint_2: motionParameters(jointSpeed=1.047198 jointAcceleration=1.396263 cartesianSpeed=0.25 cartesianAcceleration=1.2); TCP in base x=280.608 y=-116.08 z=398.046 mm, rx=-2.2371 ry=2.1464 rz=-0.0359 rad; joints [2.971, -88.172, -66.4, 247.256, 90.066, 0.681] deg
                  Folder Mouvement D
                    MoveJ speed 60 deg/s, acceleration 80 deg/s^2 (useActiveTCP=true) feature=Base
                      Waypoint Waypoint_2: motionParameters(jointSpeed=1.047198 jointAcceleration=1.396263 cartesianSpeed=0.25 cartesianAcceleration=1.2); TCP in base x=280.608 y=-116.08 z=398.046 mm, rx=-2.2371 ry=2.1464 rz=-0.0359 rad; joints [2.971, -88.172, -66.4, 247.256, 90.066, 0.681] deg
                      MoveJ speed 60 deg/s, acceleration 80 deg/s^2 (useActiveTCP=true) feature=Base
                        Waypoint Waypoint_56: TCP in base x=364.265 y=-116.054 z=192.334 mm, rx=-3.095 ry=0.0588 rz=0.0169 rad; joints [1.825, -110.55, -95.649, 295.749, 92.143, -86.362] deg
                        URCap Gripper (Robotiq_Grippers, Robotiq Inc.) dataModel(position=100.0, force=0.0, speed=0.0, positionInDouble=100.0, forceInDouble=0.0, speedInDouble=0.0, slaveIds=[2], blocking=true)
                        MoveJ speed 60 deg/s, acceleration 80 deg/s^2 (useActiveTCP=true) feature=Base
                          Waypoint Waypoint_57: TCP in base x=364.254 y=-116.07 z=333.901 mm, rx=-3.0957 ry=-0.0405 rz=0.0191 rad; joints [1.801, -106.047, -62.68, 258.123, 92.053, -89.758] deg
                          MoveJ speed 60 deg/s, acceleration 80 deg/s^2 (useActiveTCP=true) feature=Base
                            Waypoint Waypoint_58: TCP in base x=365.318 y=-268.384 z=96.47 mm, rx=-1.8274 ry=-0.0328 rz=-0.0063 rad; joints [-29.465, -175.579, 2.323, 201.363, 146.436, -157.102] deg
                            URCap Gripper (Robotiq_Grippers, Robotiq Inc.) dataModel(position=0.0, force=0.0, speed=0.0, positionInDouble=0.0, forceInDouble=0.0, speedInDouble=0.0, slaveIds=[2], blocking=true)
                            MoveJ speed 60 deg/s, acceleration 80 deg/s^2 (useActiveTCP=true) feature=Base
                              Waypoint Waypoint_2: motionParameters(jointSpeed=1.047198 jointAcceleration=1.396263 cartesianSpeed=0.25 cartesianAcceleration=1.2); TCP in base x=280.608 y=-116.08 z=398.046 mm, rx=-2.2371 ry=2.1464 rz=-0.0359 rad; joints [2.971, -88.172, -66.4, 247.256, 90.066, 0.681] deg
                              MoveJ speed 60 deg/s, acceleration 80 deg/s^2 (useActiveTCP=true) feature=Base
                                Waypoint Waypoint_56: TCP in base x=364.265 y=-116.054 z=192.334 mm, rx=-3.095 ry=0.0588 rz=0.0169 rad; joints [1.825, -110.55, -95.649, 295.749, 92.143, -86.362] deg
                                URCap Gripper (Robotiq_Grippers, Robotiq Inc.) dataModel(position=100.0, force=0.0, speed=0.0, positionInDouble=100.0, forceInDouble=0.0, speedInDouble=0.0, slaveIds=[2], blocking=true)
                                MoveJ speed 60 deg/s, acceleration 80 deg/s^2 (useActiveTCP=true) feature=Base
                                  Waypoint Waypoint_57: TCP in base x=364.254 y=-116.07 z=333.901 mm, rx=-3.0957 ry=-0.0405 rz=0.0191 rad; joints [1.801, -106.047, -62.68, 258.123, 92.053, -89.758] deg
                                  MoveJ speed 60 deg/s, acceleration 80 deg/s^2 (useActiveTCP=true) feature=Base
                                    Waypoint Waypoint_58: TCP in base x=365.318 y=-268.384 z=96.47 mm, rx=-1.8274 ry=-0.0328 rz=-0.0063 rad; joints [-29.465, -175.579, 2.323, 201.363, 146.436, -157.102] deg
                                    URCap Gripper (Robotiq_Grippers, Robotiq Inc.) dataModel(position=0.0, force=0.0, speed=0.0, positionInDouble=0.0, forceInDouble=0.0, speedInDouble=0.0, slaveIds=[2], blocking=true)
                                    MoveJ speed 60 deg/s, acceleration 80 deg/s^2 (useActiveTCP=true) feature=Base
                                      Waypoint Waypoint_2: motionParameters(jointSpeed=1.047198 jointAcceleration=1.396263 cartesianSpeed=0.25 cartesianAcceleration=1.2); TCP in base x=280.608 y=-116.08 z=398.046 mm, rx=-2.2371 ry=2.1464 rz=-0.0359 rad; joints [2.971, -88.172, -66.4, 247.256, 90.066, 0.681] deg
                                      MoveJ speed 60 deg/s, acceleration 80 deg/s^2 (useActiveTCP=true) feature=Base
                                        Waypoint Waypoint_59: TCP in base x=361.348 y=-116.091 z=193.172 mm, rx=-2.2553 ry=2.1644 rz=0.0052 rad; joints [2.324, -109.416, -97.451, 297.435, 90.248, -0.396] deg
                                        URCap Gripper (Robotiq_Grippers, Robotiq Inc.) dataModel(position=100.0, force=0.0, speed=0.0, positionInDouble=100.0, forceInDouble=0.0, speedInDouble=0.0, slaveIds=[2], blocking=true)
                                        MoveJ speed 60 deg/s, acceleration 80 deg/s^2 (useActiveTCP=true) feature=Base
                                          Waypoint Waypoint_60: TCP in base x=361.354 y=-116.078 z=193.164 mm, rx=-0.1074 ry=3.1262 rz=-0.0133 rad; joints [2.652, -109.216, -97.856, 297.904, 88.993, 88.341] deg
                                          URCap Gripper (Robotiq_Grippers, Robotiq Inc.) dataModel(position=0.0, force=0.0, speed=0.0, positionInDouble=0.0, forceInDouble=0.0, speedInDouble=0.0, slaveIds=[2], blocking=true)
                                          MoveJ speed 60 deg/s, acceleration 80 deg/s^2 (useActiveTCP=true) feature=Base
                                            Waypoint Waypoint_2: motionParameters(jointSpeed=1.047198 jointAcceleration=1.396263 cartesianSpeed=0.25 cartesianAcceleration=1.2); TCP in base x=280.608 y=-116.08 z=398.046 mm, rx=-2.2371 ry=2.1464 rz=-0.0359 rad; joints [2.971, -88.172, -66.4, 247.256, 90.066, 0.681] deg
                                            MoveJ speed 60 deg/s, acceleration 80 deg/s^2 (useActiveTCP=true) feature=Base
                                              Waypoint Waypoint_2: motionParameters(jointSpeed=1.047198 jointAcceleration=1.396263 cartesianSpeed=0.25 cartesianAcceleration=1.2); TCP in base x=280.608 y=-116.08 z=398.046 mm, rx=-2.2371 ry=2.1464 rz=-0.0359 rad; joints [2.971, -88.172, -66.4, 247.256, 90.066, 0.681] deg
                                              MoveJ speed 60 deg/s, acceleration 80 deg/s^2 (useActiveTCP=true) feature=Base
                                                Waypoint Waypoint_56: TCP in base x=364.265 y=-116.054 z=192.334 mm, rx=-3.095 ry=0.0588 rz=0.0169 rad; joints [1.825, -110.55, -95.649, 295.749, 92.143, -86.362] deg
                                                URCap Gripper (Robotiq_Grippers, Robotiq Inc.) dataModel(position=100.0, force=0.0, speed=0.0, positionInDouble=100.0, forceInDouble=0.0, speedInDouble=0.0, slaveIds=[2], blocking=true)
                                                MoveJ speed 60 deg/s, acceleration 80 deg/s^2 (useActiveTCP=true) feature=Base
                                                  Waypoint Waypoint_57: TCP in base x=364.254 y=-116.07 z=333.901 mm, rx=-3.0957 ry=-0.0405 rz=0.0191 rad; joints [1.801, -106.047, -62.68, 258.123, 92.053, -89.758] deg
                                                  MoveJ speed 60 deg/s, acceleration 80 deg/s^2 (useActiveTCP=true) feature=Base
                                                    Waypoint Waypoint_58: TCP in base x=365.318 y=-268.384 z=96.47 mm, rx=-1.8274 ry=-0.0328 rz=-0.0063 rad; joints [-29.465, -175.579, 2.323, 201.363, 146.436, -157.102] deg
                                                    URCap Gripper (Robotiq_Grippers, Robotiq Inc.) dataModel(position=0.0, force=0.0, speed=0.0, positionInDouble=0.0, forceInDouble=0.0, speedInDouble=0.0, slaveIds=[2], blocking=true)
                                                    MoveJ speed 60 deg/s, acceleration 80 deg/s^2 (useActiveTCP=true) feature=Base
                                                      Waypoint Waypoint_2: motionParameters(jointSpeed=1.047198 jointAcceleration=1.396263 cartesianSpeed=0.25 cartesianAcceleration=1.2); TCP in base x=280.608 y=-116.08 z=398.046 mm, rx=-2.2371 ry=2.1464 rz=-0.0359 rad; joints [2.971, -88.172, -66.4, 247.256, 90.066, 0.681] deg
                                                      MoveJ speed 60 deg/s, acceleration 80 deg/s^2 (useActiveTCP=true) feature=Base
                                                        Waypoint Waypoint_56: TCP in base x=364.265 y=-116.054 z=192.334 mm, rx=-3.095 ry=0.0588 rz=0.0169 rad; joints [1.825, -110.55, -95.649, 295.749, 92.143, -86.362] deg
                                                        URCap Gripper (Robotiq_Grippers, Robotiq Inc.) dataModel(position=100.0, force=0.0, speed=0.0, positionInDouble=100.0, forceInDouble=0.0, speedInDouble=0.0, slaveIds=[2], blocking=true)
                                                        MoveJ speed 60 deg/s, acceleration 80 deg/s^2 (useActiveTCP=true) feature=Base
                                                          Waypoint Waypoint_57: TCP in base x=364.254 y=-116.07 z=333.901 mm, rx=-3.0957 ry=-0.0405 rz=0.0191 rad; joints [1.801, -106.047, -62.68, 258.123, 92.053, -89.758] deg
                                                          MoveJ speed 60 deg/s, acceleration 80 deg/s^2 (useActiveTCP=true) feature=Base
                                                            Waypoint Waypoint_58: TCP in base x=365.318 y=-268.384 z=96.47 mm, rx=-1.8274 ry=-0.0328 rz=-0.0063 rad; joints [-29.465, -175.579, 2.323, 201.363, 146.436, -157.102] deg
                                                            URCap Gripper (Robotiq_Grippers, Robotiq Inc.) dataModel(position=0.0, force=0.0, speed=0.0, positionInDouble=0.0, forceInDouble=0.0, speedInDouble=0.0, slaveIds=[2], blocking=true)
                                                            MoveJ speed 60 deg/s, acceleration 80 deg/s^2 (useActiveTCP=true) feature=Base
                                                              Waypoint Waypoint_2: motionParameters(jointSpeed=1.047198 jointAcceleration=1.396263 cartesianSpeed=0.25 cartesianAcceleration=1.2); TCP in base x=280.608 y=-116.08 z=398.046 mm, rx=-2.2371 ry=2.1464 rz=-0.0359 rad; joints [2.971, -88.172, -66.4, 247.256, 90.066, 0.681] deg
                                                              Folder Mouvement D'
                                                                MoveJ speed 60 deg/s, acceleration 80 deg/s^2 (useActiveTCP=true) feature=Base
                                                                  Waypoint Waypoint_2: motionParameters(jointSpeed=1.047198 jointAcceleration=1.396263 cartesianSpeed=0.25 cartesianAcceleration=1.2); TCP in base x=280.608 y=-116.08 z=398.046 mm, rx=-2.2371 ry=2.1464 rz=-0.0359 rad; joints [2.971, -88.172, -66.4, 247.256, 90.066, 0.681] deg
                                                                  MoveJ speed 60 deg/s, acceleration 80 deg/s^2 (useActiveTCP=true) feature=Base
                                                                    Waypoint Waypoint_56: TCP in base x=364.265 y=-116.054 z=192.334 mm, rx=-3.095 ry=0.0588 rz=0.0169 rad; joints [1.825, -110.55, -95.649, 295.749, 92.143, -86.362] deg
                                                                    URCap Gripper (Robotiq_Grippers, Robotiq Inc.) dataModel(position=100.0, force=0.0, speed=0.0, positionInDouble=100.0, forceInDouble=0.0, speedInDouble=0.0, slaveIds=[2], blocking=true)
                                                                    MoveJ speed 60 deg/s, acceleration 80 deg/s^2 (useActiveTCP=true) feature=Base
                                                                      Waypoint Waypoint_57: TCP in base x=364.254 y=-116.07 z=333.901 mm, rx=-3.0957 ry=-0.0405 rz=0.0191 rad; joints [1.801, -106.047, -62.68, 258.123, 92.053, -89.758] deg
                                                                      MoveJ speed 60 deg/s, acceleration 80 deg/s^2 (useActiveTCP=true) feature=Base
                                                                        Waypoint Waypoint_58: TCP in base x=365.318 y=-268.384 z=96.47 mm, rx=-1.8274 ry=-0.0328 rz=-0.0063 rad; joints [-29.465, -175.579, 2.323, 201.363, 146.436, -157.102] deg
                                                                        URCap Gripper (Robotiq_Grippers, Robotiq Inc.) dataModel(position=0.0, force=0.0, speed=0.0, positionInDouble=0.0, forceInDouble=0.0, speedInDouble=0.0, slaveIds=[2], blocking=true)
                                                                        MoveJ speed 60 deg/s, acceleration 80 deg/s^2 (useActiveTCP=true) feature=Base
                                                                          Waypoint Waypoint_2: motionParameters(jointSpeed=1.047198 jointAcceleration=1.396263 cartesianSpeed=0.25 cartesianAcceleration=1.2); TCP in base x=280.608 y=-116.08 z=398.046 mm, rx=-2.2371 ry=2.1464 rz=-0.0359 rad; joints [2.971, -88.172, -66.4, 247.256, 90.066, 0.681] deg
                                                                          MoveJ speed 60 deg/s, acceleration 80 deg/s^2 (useActiveTCP=true) feature=Base
                                                                            Waypoint Waypoint_56: TCP in base x=364.265 y=-116.054 z=192.334 mm, rx=-3.095 ry=0.0588 rz=0.0169 rad; joints [1.825, -110.55, -95.649, 295.749, 92.143, -86.362] deg
                                                                            URCap Gripper (Robotiq_Grippers, Robotiq Inc.) dataModel(position=100.0, force=0.0, speed=0.0, positionInDouble=100.0, forceInDouble=0.0, speedInDouble=0.0, slaveIds=[2], blocking=true)
                                                                            MoveJ speed 60 deg/s, acceleration 80 deg/s^2 (useActiveTCP=true) feature=Base
                                                                              Waypoint Waypoint_57: TCP in base x=364.254 y=-116.07 z=333.901 mm, rx=-3.0957 ry=-0.0405 rz=0.0191 rad; joints [1.801, -106.047, -62.68, 258.123, 92.053, -89.758] deg
                                                                              MoveJ speed 60 deg/s, acceleration 80 deg/s^2 (useActiveTCP=true) feature=Base
                                                                                Waypoint Waypoint_58: TCP in base x=365.318 y=-268.384 z=96.47 mm, rx=-1.8274 ry=-0.0328 rz=-0.0063 rad; joints [-29.465, -175.579, 2.323, 201.363, 146.436, -157.102] deg
                                                                                URCap Gripper (Robotiq_Grippers, Robotiq Inc.) dataModel(position=0.0, force=0.0, speed=0.0, positionInDouble=0.0, forceInDouble=0.0, speedInDouble=0.0, slaveIds=[2], blocking=true)
                                                                                MoveJ speed 60 deg/s, acceleration 80 deg/s^2 (useActiveTCP=true) feature=Base
                                                                                  Waypoint Waypoint_2: motionParameters(jointSpeed=1.047198 jointAcceleration=1.396263 cartesianSpeed=0.25 cartesianAcceleration=1.2); TCP in base x=280.608 y=-116.08 z=398.046 mm, rx=-2.2371 ry=2.1464 rz=-0.0359 rad; joints [2.971, -88.172, -66.4, 247.256, 90.066, 0.681] deg
                                                                                  MoveJ speed 60 deg/s, acceleration 80 deg/s^2 (useActiveTCP=true) feature=Base
                                                                                    Waypoint Waypoint_62: TCP in base x=357.407 y=-114.5 z=192.444 mm, rx=-2.2371 ry=2.1463 rz=-0.0359 rad; joints [2.637, -108.201, -100.374, 301.253, 90.168, -0.117] deg
                                                                                    URCap Gripper (Robotiq_Grippers, Robotiq Inc.) dataModel(position=100.0, force=0.0, speed=0.0, positionInDouble=100.0, forceInDouble=0.0, speedInDouble=0.0, slaveIds=[2], blocking=true)
                                                                                    MoveJ speed 60 deg/s, acceleration 80 deg/s^2 (useActiveTCP=true) feature=Base
                                                                                      Waypoint Waypoint_61: TCP in base x=357.809 y=-114.512 z=192.818 mm, rx=-3.094 ry=-0.1205 rz=0.014 rad; joints [2.124, -109.008, -97.694, 296.22, 92.068, -92.704] deg
                                                                                      URCap Gripper (Robotiq_Grippers, Robotiq Inc.) dataModel(position=0.0, force=0.0, speed=0.0, positionInDouble=0.0, forceInDouble=0.0, speedInDouble=0.0, slaveIds=[2], blocking=true)
                                                                                      MoveJ speed 60 deg/s, acceleration 80 deg/s^2 (useActiveTCP=true) feature=Base
                                                                                        Waypoint Waypoint_2: motionParameters(jointSpeed=1.047198 jointAcceleration=1.396263 cartesianSpeed=0.25 cartesianAcceleration=1.2); TCP in base x=280.608 y=-116.08 z=398.046 mm, rx=-2.2371 ry=2.1464 rz=-0.0359 rad; joints [2.971, -88.172, -66.4, 247.256, 90.066, 0.681] deg
                                                                                        MoveJ speed 60 deg/s, acceleration 80 deg/s^2 (useActiveTCP=true) feature=Base
                                                                                          MoveJ speed 60 deg/s, acceleration 80 deg/s^2 (useActiveTCP=true) feature=Base
                                                                                            Waypoint Waypoint_56: TCP in base x=364.265 y=-116.054 z=192.334 mm, rx=-3.095 ry=0.0588 rz=0.0169 rad; joints [1.825, -110.55, -95.649, 295.749, 92.143, -86.362] deg
                                                                                            URCap Gripper (Robotiq_Grippers, Robotiq Inc.) dataModel(position=100.0, force=0.0, speed=0.0, positionInDouble=100.0, forceInDouble=0.0, speedInDouble=0.0, slaveIds=[2], blocking=true)
                                                                                            MoveJ speed 60 deg/s, acceleration 80 deg/s^2 (useActiveTCP=true) feature=Base
                                                                                              Waypoint Waypoint_57: TCP in base x=364.254 y=-116.07 z=333.901 mm, rx=-3.0957 ry=-0.0405 rz=0.0191 rad; joints [1.801, -106.047, -62.68, 258.123, 92.053, -89.758] deg
